// TwinCAT 3 PLC project kfe_rix_motion
// Title: plc-kfe-rix-motion
// Company: SLAC
// ProjectVersion: 2.8.2
// ProgramVersion: 3.1.4022.7
// CompilerDefines: K
// libraries:
//   LCLS General, * (SLAC)
//   lcls-twincat-common-components, * (SLAC)
//   lcls-twincat-motion, * (SLAC)
//   lcls-twincat-physics, * (SLAC)
//   PMPS, * (SLAC - LCLS)
//   Tc2_Standard, * (Beckhoff Automation GmbH)
//   Tc2_System, * (Beckhoff Automation GmbH)
//   Tc3_Module, * (Beckhoff Automation GmbH)
// project tree:
//   DUTs/ DUT_SATT_Filter.TcDUT, ENUM_SXR_SATT_Position.TcDUT
//   Version/ Global_Version.TcGVL
//   GVLs/ GVL.TcGVL, Main.TcGVL
//   / PlcTask.TcTTO
//   POUs/ PRG_1_PlcTask.TcPOU, PRG_2_PMPS_PRE.TcPOU, PRG_3_PMPS_POST.TcPOU, PRG_4_LOG.TcPOU, PRG_AT1K2_SOLID.TcPOU, PRG_AT2K2_SOLID.TcPOU, PRG_AT3K2_SOLID.TcPOU, PRG_IM6K2_PPM.TcPOU, PRG_LI3K2_K2B.TcPOU, PRG_PF1K2_WFS.TcPOU, PRG_LI2K2_K2A.TcPOU, PRG_IM1K1_PPM.TcPOU, PRG_AL1K2_L2SI.TcPOU, PRG_IM2K2_PPM.TcPOU, PRG_IM2K1_PPM.TcPOU, PRG_IM1K2_PPM.TcPOU, PRG_IM3K2_PPM.TcPOU, PRG_IM4K2_PPM.TcPOU, PRG_IM5K2_PPM.TcPOU, PRG_PF2K2_WFS.TcPOU, PRG_SP1K2_PAX.TcPOU, PRG_SP2K2_TXAS.TcPOU, PRG_TM1K2_ATM.TcPOU, PRG_TM2K2_ATM.TcPOU, PRG_ST3K2_TERM.TcPOU
//   POUs/TM1K2/ E_TM1K2_States.TcDUT, FB_TM1K2.TcPOU
//   POUs/TM2K2/ E_TM2K2_States.TcDUT, FB_TM2K2.TcPOU
// real-time tasks:
//   TASK PlcTask: cycle T#10ms, priority 20, ADS port 350
// motion (NC):
//   TASK NC-Task 1 SAF: cycle T#1ms, priority 4, ADS port 501
//   TASK NC-Task 1 SVB: cycle T#10ms, priority 8, ADS port 511
//   AXIS Axis 1 IM1K1-PPM-MMS (id 1)
//     Dynamic: AccelerationMaximum=200, DecelerationMaximum=200, Acceleration=200, Deceleration=200, Jerk=1000, DelayTime=0.004
//     Velo: Maximum=65
//     MotionControl: Enable=true, Range=0.0005, Time=1
//     TargetPosControl: Range=0.01, Time=1
//     OtherSettings: AllowMotionCmdToSlave=true
//     encoder EncType=29
//       EncPara: ScaleFactorNumerator=5e-05, Offset=-214686.941, MaxCount=#xffffffff, ReferenceSystem=1
//         SoftEndMinControl: Enable=true, Range=-100
//         SoftEndMaxControl: Enable=true, Range=-8.82
//         Inc: RefSoftSyncMask=#x0000ffff
//     drive DrvType=24
//       Analog: VeloReferenz=100, ScaleFactorActTorque=0.1
//       TimeComp: TaskDelayCycles=1
//     controller CtrType=2
//       CtrPara: PriorControlFactor=1
//         PosDiffControl: Range=10, Time=0.1
//         PID: PosKp=10, PosExtKp=0.01, PosExtVelo=0.0005, DeadBandPosition=0.0001
//         Observer: BandWidth=20
//   AXIS Axis 2 IM2K1-PPM-MMS (id 2)
//     Dynamic: AccelerationMaximum=200, DecelerationMaximum=200, Acceleration=200, Deceleration=200, Jerk=1000, DelayTime=0.004
//     Velo: Maximum=65
//     MotionControl: Enable=true, Range=0.0005, Time=1
//     TargetPosControl: Range=0.01, Time=1
//     OtherSettings: AllowMotionCmdToSlave=true
//     encoder EncType=29
//       EncPara: ScaleFactorNumerator=5e-05, Offset=-214686.941, MaxCount=#xffffffff, ReferenceSystem=1
//         SoftEndMinControl: Enable=true, Range=-100
//         SoftEndMaxControl: Enable=true, Range=-9.09
//         Inc: RefSoftSyncMask=#x0000ffff
//     drive DrvType=24
//       Analog: VeloReferenz=100, ScaleFactorActTorque=0.1
//       TimeComp: TaskDelayCycles=1
//     controller CtrType=2
//       CtrPara: PriorControlFactor=1
//         PosDiffControl: Range=10, Time=0.1
//         PID: PosKp=10, PosExtKp=0.01, PosExtVelo=0.0005, DeadBandPosition=0.0001
//         Observer: BandWidth=20
//   AXIS Axis 3 SPARE (id 3)
//     Velo: RefSearch=0.1, RefSync=0.1, SlowManual=0.1, FastManual=1, Maximum=1
//     OtherSettings: AllowMotionCmdToSlave=true, PulseDistancePos=1, PulseDistanceNeg=1
//     encoder EncType=29
//       EncPara: ScaleFactorNumerator=1e-06, Offset=-4264.0407, MaxCount=#xffffffff, ReferenceSystem=1
//         SoftEndMinControl: Enable=true
//         SoftEndMaxControl: Enable=true, Range=12.192
//         Inc: RefSoftSyncMask=#x0000ffff
//     drive DrvType=24
//       Analog: VeloReferenz=3.175, ScaleFactorActTorque=0.1
//       TimeComp: TaskDelayCycles=1
//     controller CtrType=1
//       CtrPara: PriorControlFactor=1
//         PosDiffControl: Range=0.1
//         Observer: BandWidth=20
//   AXIS Axis 4 IM1K2-PPM-MMS (id 4)
//     Dynamic: AccelerationMaximum=200, DecelerationMaximum=200, Acceleration=200, Deceleration=200, Jerk=500, DelayTime=0.004
//     Velo: Maximum=65
//     TargetPosControl: Range=0.002, Time=2
//     OtherSettings: AllowMotionCmdToSlave=true
//     encoder EncType=29
//       EncPara: ScaleFactorNumerator=5e-05, Offset=-214686.941, MaxCount=#xffffffff, ReferenceSystem=1
//         SoftEndMinControl: Enable=true, Range=-101
//         SoftEndMaxControl: Enable=true, Range=-9
//         Inc: RefSoftSyncMask=#x0000ffff
//     drive DrvType=24
//       Analog: VeloReferenz=100, ScaleFactorActTorque=0.1
//       TimeComp: TaskDelayCycles=1
//     controller CtrType=2
//       CtrPara: PriorControlFactor=1
//         PosDiffControl: Range=1
//         PID: PosKp=20, PosExtKp=1, PosExtVelo=0.1, DeadBandPosition=0.002
//         Observer: BandWidth=20
//   AXIS Axis 9 TM1K2-MMS-Y (id 9)
//     Dynamic: AccelerationMaximum=200, DecelerationMaximum=200, Acceleration=10, Deceleration=10, Jerk=500, DelayTime=0.004
//     Velo: Maximum=20
//     TargetPosControl: Range=0.002, Time=2
//     OtherSettings: AllowMotionCmdToSlave=true
//     encoder EncType=29
//       EncPara: ScaleFactorNumerator=5e-05, Offset=-214702, MaxCount=#xffffffff, ReferenceSystem=1
//         SoftEndMinControl: Range=-100
//         SoftEndMaxControl: Range=-16
//         Inc: RefSoftSyncMask=#x0000ffff
//     drive DrvType=24
//       Analog: VeloReferenz=100, ScaleFactorActTorque=0.1
//       TimeComp: TaskDelayCycles=1
//     controller CtrType=2
//       CtrPara: PriorControlFactor=1
//         PosDiffControl: Range=1
//         PID: PosKp=20, PosExtKp=1, PosExtVelo=0.1, DeadBandPosition=0.002
//         Observer: BandWidth=20
//   AXIS Axis 10 TM1K2-MMS-X (id 10)
//     Dynamic: AccelerationMaximum=200, DecelerationMaximum=200, Acceleration=10, Deceleration=50, Jerk=500
//     Velo: Maximum=5
//     OtherSettings: AllowMotionCmdToSlave=true
//     encoder EncType=29
//       EncPara: ScaleFactorNumerator=5e-05, MaxCount=#xffffffff, ReferenceSystem=1
//         SoftEndMinControl: Range=8.1
//         SoftEndMaxControl: Range=12.5
//         Inc: RefSoftSyncMask=#x0000ffff
//     drive DrvType=24
//       Analog: VeloReferenz=15.875, ScaleFactorActTorque=0.1
//       TimeComp: TaskDelayCycles=1
//     controller CtrType=1
//       CtrPara: PriorControlFactor=1
//         PosDiffControl: Range=0.2
//         Observer: BandWidth=20
//   AXIS Axis 6 IM2K2-PPM-MMS (id 6)
//     Dynamic: AccelerationMaximum=200, DecelerationMaximum=200, Acceleration=200, Deceleration=200, Jerk=500, DelayTime=0.004
//     Velo: Maximum=65
//     TargetPosControl: Range=0.002, Time=2
//     OtherSettings: AllowMotionCmdToSlave=true
//     encoder EncType=29
//       EncPara: ScaleFactorNumerator=5e-05, Offset=-214686.941, MaxCount=#xffffffff, ReferenceSystem=1
//         SoftEndMinControl: Enable=true, Range=-99
//         SoftEndMaxControl: Enable=true, Range=-7
//         Inc: RefSoftSyncMask=#x0000ffff
//     drive DrvType=24
//       Analog: VeloReferenz=100, ScaleFactorActTorque=0.1
//       TimeComp: TaskDelayCycles=1
//     controller CtrType=2
//       CtrPara: PriorControlFactor=1
//         PosDiffControl: Range=1
//         PID: PosKp=20, PosExtKp=1, PosExtVelo=0.1, DeadBandPosition=0.002
//         Observer: BandWidth=20
//   AXIS Axis 7 IM3K2-PPM-MMS (id 7)
//     Dynamic: AccelerationMaximum=200, DecelerationMaximum=200, Acceleration=200, Deceleration=200, Jerk=500, DelayTime=0.004
//     Velo: Maximum=65
//     TargetPosControl: Range=0.002, Time=2
//     OtherSettings: AllowMotionCmdToSlave=true
//     encoder EncType=29
//       EncPara: ScaleFactorNumerator=5e-05, Offset=-214686.941, MaxCount=#xffffffff, ReferenceSystem=1
//         SoftEndMinControl: Enable=true, Range=-108
//         SoftEndMaxControl: Enable=true, Range=-8
//         Inc: RefSoftSyncMask=#x0000ffff
//     drive DrvType=24
//       Analog: VeloReferenz=100, ScaleFactorActTorque=0.1
//       TimeComp: TaskDelayCycles=1
//     controller CtrType=2
//       CtrPara: PriorControlFactor=1
//         PosDiffControl: Range=1
//         PID: PosKp=20, PosExtKp=1, PosExtVelo=0.1, DeadBandPosition=0.002
//         Observer: BandWidth=20
//   AXIS Axis 8 IM4K2-PPM-MMS (id 8)
//     Dynamic: AccelerationMaximum=200, DecelerationMaximum=200, Acceleration=200, Deceleration=200, Jerk=1000, DelayTime=0.004
//     Velo: Maximum=65
//     MotionControl: Enable=true, Range=0.0005, Time=1
//     TargetPosControl: Range=0.01, Time=1
//     OtherSettings: AllowMotionCmdToSlave=true
//     encoder EncType=29
//       EncPara: ScaleFactorNumerator=5e-05, Offset=-214686.941, MaxCount=#xffffffff, ReferenceSystem=1
//         SoftEndMinControl: Enable=true, Range=-100
//         SoftEndMaxControl: Enable=true, Range=-10
//         Inc: RefSoftSyncMask=#x0000ffff
//     drive DrvType=24
//       Analog: VeloReferenz=100, ScaleFactorActTorque=0.1
//       TimeComp: TaskDelayCycles=1
//     controller CtrType=2
//       CtrPara: PriorControlFactor=1
//         PosDiffControl: Range=10, Time=0.1
//         PID: PosKp=10, PosExtKp=0.01, PosExtVelo=0.0005, DeadBandPosition=0.0001
//         Observer: BandWidth=20
//   AXIS Axis 14 IM5K2-PPM-MMS (id 14)
//     Dynamic: AccelerationMaximum=200, DecelerationMaximum=200, Acceleration=200, Deceleration=200, Jerk=1000, DelayTime=0.004
//     Velo: Maximum=65
//     MotionControl: Enable=true, Range=0.0005, Time=1
//     TargetPosControl: Range=0.01, Time=1
//     OtherSettings: AllowMotionCmdToSlave=true
//     encoder EncType=29
//       EncPara: ScaleFactorNumerator=5e-05, Offset=-214686.941, MaxCount=#xffffffff, ReferenceSystem=1
//         SoftEndMinControl: Enable=true, Range=-100
//         SoftEndMaxControl: Enable=true, Range=-8
//         Inc: RefSoftSyncMask=#x0000ffff
//     drive DrvType=24
//       Analog: VeloReferenz=100, ScaleFactorActTorque=0.1
//       TimeComp: TaskDelayCycles=1
//     controller CtrType=2
//       CtrPara: PriorControlFactor=1
//         PosDiffControl: Range=10, Time=0.1
//         PID: PosKp=10, PosExtKp=0.01, PosExtVelo=0.0005, DeadBandPosition=0.0001
//         Observer: BandWidth=20
//   AXIS Axis 5 AL1K2-L2SI-MMS (id 5)
//     Dynamic: AccelerationMaximum=200, DecelerationMaximum=200, Acceleration=200, Deceleration=200, Jerk=500, DelayTime=0.004
//     Velo: Maximum=10
//     TargetPosControl: Range=0.002, Time=2
//     OtherSettings: AllowMotionCmdToSlave=true
//     encoder EncType=29
//       EncPara: ScaleFactorNumerator=5e-05, Offset=-214686.941, MaxCount=#xffffffff, ReferenceSystem=1
//         SoftEndMinControl: Range=-108.74
//         SoftEndMaxControl: Range=-33.49
//         Inc: RefSoftSyncMask=#x0000ffff
//     drive DrvType=24
//       Analog: VeloReferenz=100, ScaleFactorActTorque=0.1
//       TimeComp: TaskDelayCycles=1
//     controller CtrType=2
//       CtrPara: PriorControlFactor=1
//         PosDiffControl: Range=1
//         PID: PosKp=20, PosExtKp=1, PosExtVelo=0.1, DeadBandPosition=0.002
//         Observer: BandWidth=20
//   AXIS Axis 11 LI2K2-K2A_OUT-MMS (id 11)
//     Dynamic: AccelerationMaximum=200, DecelerationMaximum=200, Acceleration=200, Deceleration=200, Jerk=500, DelayTime=0.004
//     Velo: Maximum=65
//     TargetPosControl: Range=0.002, Time=2
//     OtherSettings: AllowMotionCmdToSlave=true
//     encoder EncType=29
//       EncPara: ScaleFactorNumerator=5e-05, Offset=-214680, MaxCount=#xffffffff, ReferenceSystem=1
//         SoftEndMinControl: Range=-107.43
//         SoftEndMaxControl: Range=1.35
//         Inc: RefSoftSyncMask=#x0000ffff
//     drive DrvType=24
//       Analog: VeloReferenz=100, ScaleFactorActTorque=0.1
//       TimeComp: TaskDelayCycles=1
//     controller CtrType=2
//       CtrPara: PriorControlFactor=1
//         PosDiffControl: Range=1
//         PID: PosKp=20, PosExtKp=1, PosExtVelo=0.1, DeadBandPosition=0.002
//         Observer: BandWidth=20
//   AXIS Axis 12 PF1K2-WFS-MMS-Y (id 12)
//     Dynamic: AccelerationMaximum=200, DecelerationMaximum=200, Acceleration=10, Deceleration=10, Jerk=500, DelayTime=0.004
//     Velo: Maximum=20
//     TargetPosControl: Range=0.002, Time=2
//     OtherSettings: AllowMotionCmdToSlave=true
//     encoder EncType=29
//       EncPara: ScaleFactorNumerator=5e-05, Offset=-214679, MaxCount=#xffffffff, ReferenceSystem=1
//         SoftEndMinControl: Enable=true, Range=-94
//         SoftEndMaxControl: Enable=true, Range=-9.71
//         Inc: RefSoftSyncMask=#x0000ffff
//     drive DrvType=24
//       Analog: VeloReferenz=100, ScaleFactorActTorque=0.1
//       TimeComp: TaskDelayCycles=1
//     controller CtrType=2
//       CtrPara: PriorControlFactor=1
//         PosDiffControl: Range=1
//         PID: PosKp=20, PosExtKp=1, PosExtVelo=0.1, DeadBandPosition=0.002
//         Observer: BandWidth=20
//   AXIS Axis 13 PF1K2-WFS-MMS-Z (id 13)
//     Dynamic: AccelerationMaximum=200, DecelerationMaximum=200, Acceleration=10, Deceleration=50, Jerk=500
//     Velo: Maximum=5
//     OtherSettings: AllowMotionCmdToSlave=true
//     encoder EncType=29
//       EncPara: ScaleFactorNumerator=5e-05, MaxCount=#xffffffff, ReferenceSystem=1
//         SoftEndMinControl: Range=6.5
//         SoftEndMaxControl: Range=56
//         Inc: RefSoftSyncMask=#x0000ffff
//     drive DrvType=24
//       DrvPara: Inverse=true
//         Analog: VeloReferenz=15.875, ScaleFactorActTorque=0.1
//         TimeComp: TaskDelayCycles=1
//     controller CtrType=1
//       CtrPara: PriorControlFactor=1
//         PosDiffControl: Range=1
//         Observer: BandWidth=20
//   AXIS Axis 15 TM2K2-MMS-Y (id 15)
//     Dynamic: AccelerationMaximum=200, DecelerationMaximum=200, Acceleration=10, Deceleration=10, Jerk=500, DelayTime=0.004
//     Velo: Maximum=20
//     TargetPosControl: Range=0.002, Time=2
//     OtherSettings: AllowMotionCmdToSlave=true
//     encoder EncType=29
//       EncPara: ScaleFactorNumerator=5e-05, Offset=-214682, MaxCount=#xffffffff, ReferenceSystem=1
//         SoftEndMinControl: Range=-100
//         SoftEndMaxControl: Range=-16
//         Inc: RefSoftSyncMask=#x0000ffff
//     drive DrvType=24
//       Analog: VeloReferenz=100, ScaleFactorActTorque=0.1
//       TimeComp: TaskDelayCycles=1
//     controller CtrType=2
//       CtrPara: PriorControlFactor=1
//         PosDiffControl: Range=1
//         PID: PosKp=20, PosExtKp=1, PosExtVelo=0.1, DeadBandPosition=0.002
//         Observer: BandWidth=20
//   AXIS Axis 16 TM2K2-MMS-X (id 16)
//     Dynamic: AccelerationMaximum=200, DecelerationMaximum=200, Acceleration=10, Deceleration=50, Jerk=500
//     Velo: Maximum=5
//     OtherSettings: AllowMotionCmdToSlave=true
//     encoder EncType=29
//       EncPara: ScaleFactorNumerator=5e-05, MaxCount=#xffffffff, ReferenceSystem=1
//         SoftEndMinControl: Enable=true, Range=16.5
//         SoftEndMaxControl: Enable=true, Range=21
//         Inc: RefSoftSyncMask=#x0000ffff
//     drive DrvType=24
//       DrvPara: Inverse=true
//         Analog: VeloReferenz=15.875, ScaleFactorActTorque=0.1
//         TimeComp: TaskDelayCycles=1
//     controller CtrType=1
//       CtrPara: PriorControlFactor=1
//         PosDiffControl: Range=0.2
//         Observer: BandWidth=20
//   AXIS Axis 17 AT2K2-SOLID-MMS-01 (id 17)
//     Dynamic: AccelerationMaximum=400, DecelerationMaximum=400, Acceleration=160, Deceleration=160, Jerk=80, DelayTime=0.008
//     Velo: SlowManual=1, FastManual=10, Maximum=80
//     OtherSettings: AllowMotionCmdToSlave=true
//     encoder EncType=29
//       EncPara: ScaleFactorNumerator=5e-05, MaxCount=#xffffffff
//         SoftEndMinControl: Enable=true, Range=16.5
//         SoftEndMaxControl: Enable=true, Range=152.5
//         Inc: RefSoftSyncMask=#x0000ffff
//     drive DrvType=24
//       Analog: VeloReferenz=40, ScaleFactorActTorque=0.1
//       TimeComp: TaskDelayCycles=1
//     controller CtrType=2
//       CtrPara: PriorControlFactor=1
//         PosDiffControl: Range=0.2
//         PID: PosKp=20, PosExtKp=20, PosExtVelo=0.1, DeadBandPosition=0.01
//         Observer: BandWidth=20
//   AXIS Axis 18 AT2K2-SOLID-MMS-02 (id 18)
//     Dynamic: AccelerationMaximum=400, DecelerationMaximum=400, Acceleration=160, Deceleration=160, Jerk=80, DelayTime=0.008
//     Velo: SlowManual=1, FastManual=5, Maximum=80
//     OtherSettings: AllowMotionCmdToSlave=true
//     encoder EncType=29
//       EncPara: ScaleFactorNumerator=5e-05, MaxCount=#xffffffff
//         SoftEndMinControl: Enable=true, Range=17.5
//         SoftEndMaxControl: Enable=true, Range=152.5
//         Inc: RefSoftSyncMask=#x0000ffff
//     drive DrvType=24
//       Analog: VeloReferenz=40, ScaleFactorActTorque=0.1
//       TimeComp: TaskDelayCycles=1
//     controller CtrType=2
//       CtrPara: PriorControlFactor=1
//         PosDiffControl: Range=0.2
//         PID: PosKp=20, PosExtKp=20, PosExtVelo=0.1, DeadBandPosition=0.01
//         Observer: BandWidth=20
//   AXIS Axis 19 AT2K2-SOLID-MMS-03 (id 19)
//     Dynamic: AccelerationMaximum=400, DecelerationMaximum=400, Acceleration=160, Deceleration=160, Jerk=80, DelayTime=0.008
//     Velo: SlowManual=1, FastManual=10, Maximum=80
//     OtherSettings: AllowMotionCmdToSlave=true
//     encoder EncType=29
//       EncPara: ScaleFactorNumerator=5e-05, MaxCount=#xffffffff
//         SoftEndMinControl: Enable=true, Range=16.5
//         SoftEndMaxControl: Enable=true, Range=152.5
//         Inc: RefSoftSyncMask=#x0000ffff
//     drive DrvType=24
//       Analog: VeloReferenz=40, ScaleFactorActTorque=0.1
//       TimeComp: TaskDelayCycles=1
//     controller CtrType=2
//       CtrPara: PriorControlFactor=1
//         PosDiffControl: Range=0.2
//         PID: PosKp=20, PosExtKp=20, PosExtVelo=0.1, DeadBandPosition=0.01
//         Observer: BandWidth=20
//   AXIS Axis 20 AT2K2-SOLID-MMS-04 (id 20)
//     Dynamic: AccelerationMaximum=400, DecelerationMaximum=400, Acceleration=160, Deceleration=160, Jerk=80, DelayTime=0.008
//     Velo: SlowManual=1, FastManual=10, Maximum=80
//     OtherSettings: AllowMotionCmdToSlave=true
//     encoder EncType=29
//       EncPara: ScaleFactorNumerator=5e-05, MaxCount=#xffffffff
//         SoftEndMinControl: Enable=true, Range=17.8
//         SoftEndMaxControl: Enable=true, Range=152.5
//         Inc: RefSoftSyncMask=#x0000ffff
//     drive DrvType=24
//       Analog: VeloReferenz=40, ScaleFactorActTorque=0.1
//       TimeComp: TaskDelayCycles=1
//     controller CtrType=2
//       CtrPara: PriorControlFactor=1
//         PosDiffControl: Range=0.2
//         PID: PosKp=20, PosExtKp=20, PosExtVelo=0.1, DeadBandPosition=0.01
//         Observer: BandWidth=20
//   AXIS Axis 21 LI3K2-K2B-MMS (id 21)
//     Dynamic: AccelerationMaximum=200, DecelerationMaximum=200, Acceleration=200, Deceleration=200, Jerk=500, DelayTime=0.004
//     Velo: Maximum=65
//     TargetPosControl: Range=0.002, Time=2
//     OtherSettings: AllowMotionCmdToSlave=true
//     encoder EncType=29
//       EncPara: ScaleFactorNumerator=5e-05, Offset=-214687, MaxCount=#xffffffff, ReferenceSystem=1
//         SoftEndMinControl: Enable=true, Range=-107.43
//         SoftEndMaxControl: Enable=true, Range=1.35
//         Inc: RefSoftSyncMask=#x0000ffff
//     drive DrvType=24
//       Analog: VeloReferenz=100, ScaleFactorActTorque=0.1
//       TimeComp: TaskDelayCycles=1
//     controller CtrType=2
//       CtrPara: PriorControlFactor=1
//         PosDiffControl: Range=1
//         PID: PosKp=20, PosExtKp=1, PosExtVelo=0.1, DeadBandPosition=0.002
//         Observer: BandWidth=20
//   AXIS Axis 22 PF2K2-WFS-MMS-Y (id 22)
//     Dynamic: AccelerationMaximum=200, DecelerationMaximum=200, Acceleration=10, Deceleration=10, Jerk=500, DelayTime=0.004
//     Velo: Maximum=20
//     TargetPosControl: Range=0.002, Time=2
//     OtherSettings: AllowMotionCmdToSlave=true
//     encoder EncType=29
//       EncPara: ScaleFactorNumerator=5e-05, Offset=-214687, MaxCount=#xffffffff, ReferenceSystem=1
//         SoftEndMinControl: Enable=true, Range=-99.33
//         SoftEndMaxControl: Enable=true, Range=-9.71
//         Inc: RefSoftSyncMask=#x0000ffff
//     drive DrvType=24
//       Analog: VeloReferenz=100, ScaleFactorActTorque=0.1
//       TimeComp: TaskDelayCycles=1
//     controller CtrType=2
//       CtrPara: PriorControlFactor=1
//         PosDiffControl: Range=1
//         PID: PosKp=20, PosExtKp=1, PosExtVelo=0.1, DeadBandPosition=0.002
//         Observer: BandWidth=20
//   AXIS Axis 23 PF2K2-WFS-MMS-Z (id 23)
//     Dynamic: AccelerationMaximum=200, DecelerationMaximum=200, Acceleration=10, Deceleration=50, Jerk=500
//     Velo: Maximum=5
//     OtherSettings: AllowMotionCmdToSlave=true
//     encoder EncType=29
//       EncPara: ScaleFactorNumerator=5e-05, MaxCount=#xffffffff, ReferenceSystem=1
//         SoftEndMinControl: Range=6.5
//         SoftEndMaxControl: Range=56
//         Inc: RefSoftSyncMask=#x0000ffff
//     drive DrvType=24
//       DrvPara: Inverse=true
//         Analog: VeloReferenz=15.875, ScaleFactorActTorque=0.1
//         TimeComp: TaskDelayCycles=1
//     controller CtrType=1
//       CtrPara: PriorControlFactor=1
//         PosDiffControl: Range=1
//         PID: PosKp=10
//         Observer: BandWidth=20
//   AXIS Axis 24 IM6K2-PPM-MMS (id 24)
//     Dynamic: AccelerationMaximum=200, DecelerationMaximum=200, Acceleration=200, Deceleration=200, Jerk=1000, DelayTime=0.004
//     Velo: Maximum=65
//     MotionControl: Enable=true, Range=0.0005, Time=1
//     TargetPosControl: Range=0.01, Time=1
//     OtherSettings: AllowMotionCmdToSlave=true
//     encoder EncType=29
//       EncPara: ScaleFactorNumerator=5e-05, Offset=-214686.941, MaxCount=#xffffffff, ReferenceSystem=1
//         SoftEndMinControl: Enable=true, Range=-100
//         SoftEndMaxControl: Enable=true, Range=-8
//         Inc: RefSoftSyncMask=#x0000ffff
//     drive DrvType=24
//       Analog: VeloReferenz=100, ScaleFactorActTorque=0.1
//       TimeComp: TaskDelayCycles=1
//     controller CtrType=2
//       CtrPara: PriorControlFactor=1
//         PosDiffControl: Range=10, Time=0.1
//         PID: PosKp=10, PosExtKp=0.01, PosExtVelo=0.0005, DeadBandPosition=0.0001
//         Observer: BandWidth=20
//   AXIS Axis 25 AT1K2-SOLID-MMS-01 (id 25)
//     Dynamic: AccelerationMaximum=400, DecelerationMaximum=400, Acceleration=160, Deceleration=160, Jerk=80, DelayTime=0.008
//     Velo: SlowManual=1, FastManual=10, Maximum=80
//     OtherSettings: AllowMotionCmdToSlave=true
//     encoder EncType=29
//       EncPara: ScaleFactorNumerator=5e-05, MaxCount=#xffffffff
//         SoftEndMinControl: Enable=true, Range=19
//         SoftEndMaxControl: Enable=true, Range=152.2
//         Inc: RefSoftSyncMask=#x0000ffff
//     drive DrvType=24
//       Analog: VeloReferenz=40, ScaleFactorActTorque=0.1
//       TimeComp: TaskDelayCycles=1
//     controller CtrType=2
//       CtrPara: PriorControlFactor=1
//         PosDiffControl: Range=0.2
//         PID: PosKp=20, PosExtKp=20, PosExtVelo=0.1, DeadBandPosition=0.01
//         Observer: BandWidth=20
//   AXIS Axis 26 AT1K2-SOLID-MMS-02 (id 26)
//     Dynamic: AccelerationMaximum=400, DecelerationMaximum=400, Acceleration=160, Deceleration=160, Jerk=80, DelayTime=0.008
//     Velo: SlowManual=1, FastManual=10, Maximum=80
//     OtherSettings: AllowMotionCmdToSlave=true
//     encoder EncType=29
//       EncPara: ScaleFactorNumerator=5e-05, MaxCount=#xffffffff
//         SoftEndMinControl: Enable=true, Range=19
//         SoftEndMaxControl: Enable=true, Range=152.2
//         Inc: RefSoftSyncMask=#x0000ffff
//     drive DrvType=24
//       Analog: VeloReferenz=40, ScaleFactorActTorque=0.1
//       TimeComp: TaskDelayCycles=1
//     controller CtrType=2
//       CtrPara: PriorControlFactor=1
//         PosDiffControl: Range=0.2
//         PID: PosKp=20, PosExtKp=20, PosExtVelo=0.1, DeadBandPosition=0.01
//         Observer: BandWidth=20
//   AXIS Axis 27 AT1K2-SOLID-MMS-03 (id 27)
//     Dynamic: AccelerationMaximum=400, DecelerationMaximum=400, Acceleration=160, Deceleration=160, Jerk=80, DelayTime=0.008
//     Velo: SlowManual=1, FastManual=10, Maximum=6
//     OtherSettings: AllowMotionCmdToSlave=true
//     encoder EncType=29
//       EncPara: ScaleFactorNumerator=5e-05, MaxCount=#xffffffff
//         SoftEndMinControl: Enable=true, Range=23
//         SoftEndMaxControl: Enable=true, Range=67
//         Inc: RefSoftSyncMask=#x0000ffff
//     drive DrvType=24
//       Analog: VeloReferenz=2.5, ScaleFactorActTorque=0.1
//       TimeComp: TaskDelayCycles=1
//     controller CtrType=2
//       CtrPara: PriorControlFactor=1
//         PosDiffControl: Range=0.2
//         PID: PosKp=5, PosExtKp=5, PosExtVelo=0.1, DeadBandPosition=0.001
//         Observer: BandWidth=20
//   AXIS Axis 37 SP1K2-PAX-BB-MMS-Y-02 (id 37)
//     Velo: SlowManual=0.5, FastManual=1, Maximum=1.5
//     OtherSettings: AllowMotionCmdToSlave=true
//     encoder EncType=29
//       EncPara: ScaleFactorNumerator=0.000244, Offset=-8917.43869, MaxCount=#xffffffff
//         SoftEndMinControl: Enable=true
//         SoftEndMaxControl: Enable=true, Range=43
//         Inc: RefSoftSyncMask=#x0000ffff
//     drive DrvType=24
//       DrvPara: Inverse=true
//         Analog: VeloReferenz=2.5, ScaleFactorActTorque=0.1
//         TimeComp: TaskDelayCycles=1
//     controller CtrType=1
//       CtrPara: PriorControlFactor=1
//         Observer: BandWidth=20
//   AXIS Axis 36 SP1K2-PAX-BB-MMS-Y-01 (id 36)
//     Velo: SlowManual=0.5, FastManual=1, Maximum=1.5
//     OtherSettings: AllowMotionCmdToSlave=true
//     encoder EncType=29
//       EncPara: ScaleFactorNumerator=0.000244, Offset=-1039158.545, MaxCount=#xffffffff
//         SoftEndMinControl: Enable=true, Range=-43
//         SoftEndMaxControl: Enable=true
//         Inc: RefSoftSyncMask=#x0000ffff
//     drive DrvType=24
//       Analog: VeloReferenz=2.5, ScaleFactorActTorque=0.1
//       TimeComp: TaskDelayCycles=1
//     controller CtrType=1
//       CtrPara: PriorControlFactor=1
//         Observer: BandWidth=20
//   AXIS Axis 35 SP1K2-PAX-TAR-MMS-RY (id 35)
//     OtherSettings: AllowMotionCmdToSlave=true
//     encoder EncType=1
//       Inc: RefSoftSyncMask=#x0000ffff
//     drive DrvType=5
//       Analog: ScaleFactorActTorque=0.1
//       TimeComp: TaskDelayCycles=1
//     controller CtrType=1
//       CtrPara: PriorControlFactor=1
//         Observer: BandWidth=20
//   AXIS Axis 34 SP1K2-PAX-TAR-MMS-Z (id 34)
//     Velo: SlowManual=0.1, FastManual=1, Maximum=1
//     OtherSettings: AllowMotionCmdToSlave=true
//     encoder EncType=29
//       EncPara: ScaleFactorNumerator=0.000244, Offset=-15736.2402, MaxCount=#xffffffff
//         SoftEndMinControl: Enable=true
//         Inc: RefSoftSyncMask=#x0000ffff
//     drive DrvType=24
//       Analog: VeloReferenz=2, ScaleFactorActTorque=0.1
//       TimeComp: TaskDelayCycles=1
//     controller CtrType=1
//       CtrPara: PriorControlFactor=1
//         Observer: BandWidth=20
//   AXIS Axis 33 SP1K2-PAX-TAR-MMS-Y (id 33)
//     Velo: SlowManual=0.5, FastManual=1, Maximum=1
//     OtherSettings: AllowMotionCmdToSlave=true
//     encoder EncType=29
//       EncPara: ScaleFactorNumerator=5e-05, MaxCount=#xffffffff
//         Inc: RefSoftSyncMask=#x0000ffff
//     drive DrvType=24
//       DrvPara: Inverse=true
//         Analog: VeloReferenz=2, ScaleFactorActTorque=0.1
//         TimeComp: TaskDelayCycles=1
//     controller CtrType=1
//       CtrPara: PriorControlFactor=1
//         Observer: BandWidth=20
//   AXIS Axis 32 SP1K2-PAX-TAR-MMS-X (id 32)
//     Dynamic: AccelerationMaximum=1, DecelerationMaximum=1
//     Velo: SlowManual=0.1, FastManual=1, Maximum=0.5
//     OtherSettings: AllowMotionCmdToSlave=true
//     encoder EncType=29
//       EncPara: ScaleFactorNumerator=0.000244, Offset=-15554.7601, MaxCount=#xffffffff
//         Inc: RefSoftSyncMask=#x0000ffff
//     drive DrvType=24
//       DrvPara: Inverse=true
//         Analog: VeloReferenz=12.5, ScaleFactorActTorque=0.1
//         TimeComp: TaskDelayCycles=1
//     controller CtrType=1
//       CtrPara: PriorControlFactor=1
//         Observer: BandWidth=20
//   AXIS Axis 31 SP1K2-PAX-FRAME-MMS-X (id 31)
//     Dynamic: AccelerationMaximum=1500
//     Velo: Maximum=1
//     OtherSettings: AllowMotionCmdToSlave=true
//     encoder EncType=29
//       EncPara: ScaleFactorNumerator=5e-05, MaxCount=#xffffffff
//         Inc: RefSoftSyncMask=#x0000ffff
//     drive DrvType=24
//       Analog: VeloReferenz=10, ScaleFactorActTorque=0.1
//       TimeComp: TaskDelayCycles=1
//     controller CtrType=1
//       CtrPara: PriorControlFactor=1
//         Observer: BandWidth=20
//   AXIS Axis 30 SP1K2-PAX-FRAME-MMS-Y-03 (id 30)
//     Velo: Maximum=1
//     OtherSettings: AllowMotionCmdToSlave=true
//     encoder EncType=29
//       EncPara: ScaleFactorNumerator=5e-05, MaxCount=#xffffffff
//         Inc: RefSoftSyncMask=#x0000ffff
//     drive DrvType=24
//       Analog: VeloReferenz=2.5, ScaleFactorActTorque=0.1
//       TimeComp: TaskDelayCycles=1
//     controller CtrType=1
//       CtrPara: PriorControlFactor=1
//         Observer: BandWidth=20
//   AXIS Axis 29 SP1K2-PAX-FRAME-MMS-Y-02 (id 29)
//     Velo: Maximum=1
//     OtherSettings: AllowMotionCmdToSlave=true
//     encoder EncType=29
//       EncPara: ScaleFactorNumerator=5e-05, MaxCount=#xffffffff
//         Inc: RefSoftSyncMask=#x0000ffff
//     drive DrvType=24
//       Analog: VeloReferenz=2.5, ScaleFactorActTorque=0.1
//       TimeComp: TaskDelayCycles=1
//     controller CtrType=1
//       CtrPara: PriorControlFactor=1
//         Observer: BandWidth=20
//   AXIS Axis 28 SP1K2-PAX-FRAME-MMS-Y-01 (id 28)
//     Velo: Maximum=1
//     OtherSettings: AllowMotionCmdToSlave=true
//     encoder EncType=29
//       EncPara: ScaleFactorNumerator=5e-06, MaxCount=#xffffffff
//         Inc: RefSoftSyncMask=#x0000ffff
//     drive DrvType=24
//       Analog: VeloReferenz=2.5, ScaleFactorActTorque=0.1
//       TimeComp: TaskDelayCycles=1
//     controller CtrType=1
//       CtrPara: PriorControlFactor=1
//         Observer: BandWidth=20
// I/O:
//   DEVICE PLC Rail (EtherCAT), AmsNetId 172.21.140.70.2.1
//     Power (EK1200) [EK1200-5000 EtherCAT Power supply (2A E-Bus)]
//       License (EL6070)
//       PMPS_FFO [EL2202 2Ch. Dig. Output 24V, 0.5A]
//       PMPS_PRE [EL6695 EtherCAT Bridge terminal (Primary)]
//       Fiber Coupler (EK1521-0010) [EK1521-0010 1 port EtherCAT junction (FX-SingleMode)]
//         Term 34 (EK1501-0010) [EK1501-0010 EtherCAT Coupler (2A E-Bus, FX-SingleMode, ID switch)]
//           Term 35 (EL9410) [EL9410 E-Bus Power Supplier  (Diagnostics)]
//           Term 36 (EL2202) [EL2202 2Ch. Dig. Output 24V, 0.5A]
//           Term 37 (EL6070) [EL6070 1Ch. Licensing-Terminal]
//           Term 38 (EL6695) [EL6695 EtherCAT Bridge terminal (Primary)]
//           Term 39 (EK1122) [EK1122 2 port EtherCAT junction]
//             IM1K2-PPM (EK1100) [EK1100 EtherCAT Coupler (2A E-Bus)]
//               IM1K2-EL7041-E1 [EL7041 1Ch. Stepper motor output stage (50V, 5A)]
//               IM1K2-EL5042-E2 [EL5042 2Ch. BiSS-C Encoder]
//               IM1K2-EL2004-E3 [EL2004 4Ch. Dig. Output 24V, 0.5A]
//               IM1K2-EL3314-E4 [EL3314 4Ch. Ana. Input Thermocouple (TC)]
//               IM1K2-EL3052-E5 [EL3052 2Ch. Ana. Input 4-20mA]
//               IM1K2-EL3062-E6 [EL3062 2Ch. Ana. Input 0-10V]
//               IM1K2-EL4004-E7 [EL4004 4Ch. Ana. Output 0-10V, 12bit]
//               IM1K2-EL9011-E8 [EL9011 End Terminal]
//             AL1K2-L2SI (EK1100) [EK1100 EtherCAT Coupler (2A E-Bus)]
//               AL1K2-EL7041-E1 [EL7041 1Ch. Stepper motor output stage (50V, 5A)]
//               AL1K2-EL5042-E2 [EL5042 2Ch. BiSS-C Encoder]
//               AL1K2-EL2004-E3 [EL2004 4Ch. Dig. Output 24V, 0.5A]
//               AL1K2-EL4004-E4 [EL4004 4Ch. Ana. Output 0-10V, 12bit]
//               AL1K2-EL9011-E5 [EL9011 End Terminal]
//           Term 49 (EK1122) [EK1122 2 port EtherCAT junction]
//             IM2K2-PPM (EK1100) [EK1100 EtherCAT Coupler (2A E-Bus)]
//               IM2K2-EL7041-E1 [EL7041 1Ch. Stepper motor output stage (50V, 5A)]
//               IM2K2-EL5042-E2 [EL5042 2Ch. BiSS-C Encoder]
//               IM2K2-EL2004-E3 [EL2004 4Ch. Dig. Output 24V, 0.5A]
//               IM2K2-EL3314-E4 [EL3314 4Ch. Ana. Input Thermocouple (TC)]
//               IM2K2-EL3052-E5 [EL3052 2Ch. Ana. Input 4-20mA]
//               IM2K2-EL3062-E6 [EL3062 2Ch. Ana. Input 0-10V]
//               IM2K2-EL4004-E7 [EL4004 4Ch. Ana. Output 0-10V, 12bit]
//               IM2K2-EL9011-E8
//           Term 50 (EK1122) [EK1122 2 port EtherCAT junction]
//             IM3K2-PPM (EK1100) [EK1100 EtherCAT Coupler (2A E-Bus)]
//               IM3K2-EL7041-E1 [EL7041 1Ch. Stepper motor output stage (50V, 5A)]
//               IM3K2-EL5042-E2 [EL5042 2Ch. BiSS-C Encoder]
//               IM3K2-EL2004-E3 [EL2004 4Ch. Dig. Output 24V, 0.5A]
//               IM3K2-EL3314-E4 [EL3314 4Ch. Ana. Input Thermocouple (TC)]
//               IM3K2-EL3052-E5 [EL3052 2Ch. Ana. Input 4-20mA]
//               IM3K2-EL3062-E6 [EL3062 2Ch. Ana. Input 0-10V]
//               IM3K2-EL4004-E7 [EL4004 4Ch. Ana. Output 0-10V, 12bit]
//               IM3K2-EL9011-E8
//             IM4K2-PPM (EK1100) [EK1100 EtherCAT Coupler (2A E-Bus)]
//               IM4K2-EL7041-E1 [EL7041 1Ch. Stepper motor output stage (50V, 5A)]
//               IM4K2-EL5042-E2 [EL5042 2Ch. BiSS-C Encoder]
//               IM4K2-EL2004-E3 [EL2004 4Ch. Dig. Output 24V, 0.5A]
//               IM4K2-EL3314-E4 [EL3314 4Ch. Ana. Input Thermocouple (TC)]
//               IM4K2-EL3052-E5 [EL3052 2Ch. Ana. Input 4-20mA]
//               IM4K2-EL3062-E6 [EL3062 2Ch. Ana. Input 0-10V]
//               IM4K2-EL4004-E7 [EL4004 4Ch. Ana. Output 0-10V, 12bit]
//               IM4K2-EL3602-0002-E8 [EL3602-0002 2Ch. Ana. Input +/-200mV, Diff. 24bit]
//               IM4K2-EL9011-E9 [EL9011 End Terminal]
//           Term 51 (EK1110)
//         Term 123 (EK1100) [EK1100 EtherCAT Coupler (2A E-Bus)]
//           Term 124 (EK1122) [EK1122 2 port EtherCAT junction]
//             TM1K2-K2A (EK1100) [EK1100 EtherCAT Coupler (2A E-Bus)]
//               TM1K2-EL7041-E1 [EL7041 1Ch. Stepper motor output stage (50V, 5A)]
//               TM1K2-EL7041-E2 [EL7041 1Ch. Stepper motor output stage (50V, 5A)]
//               TM1K2-EL5042-E3 [EL5042 2Ch. BiSS-C Encoder]
//               TM1K2-EL2004-E4 [EL2004 4Ch. Dig. Output 24V, 0.5A]
//               TM1K2-EL3314-E5 [EL3314 4Ch. Ana. Input Thermocouple (TC)]
//               TM1K2-EL9011-E6 [EL9011 End Terminal]
//           Term 131 (EK1122) [EK1122 2 port EtherCAT junction]
//             LI2K2-K2A_OUT  (EK1100) [EK1100 EtherCAT Coupler (2A E-Bus)]
//               LI2K2-EL7041-E1 [EL7041 1Ch. Stepper motor output stage (50V, 5A)]
//               LI2K2-EL2004-E2 [EL2004 4Ch. Dig. Output 24V, 0.5A]
//               LI2K2-EL5042-E3 [EL5042 2Ch. BiSS-C Encoder]
//               LI2K2-EL9011-E4 [EL9011 End Terminal]
//             PF1K2-WFS (EK1100) [EK1100 EtherCAT Coupler (2A E-Bus)]
//               PF1K2-EL7041-E1 [EL7041 1Ch. Stepper motor output stage (50V, 5A)]
//               PF1K2-EL7041-E2 [EL7041 1Ch. Stepper motor output stage (50V, 5A)]
//               PF1K2-EL5042-E3 [EL5042 2Ch. BiSS-C Encoder]
//               PF1K2-EL2004-E4 [EL2004 4Ch. Dig. Output 24V, 0.5A]
//               PF1K2-EL3314-E5 [EL3314 4Ch. Ana. Input Thermocouple (TC)]
//               PF1K2-EL9011-E6 [EL9011 End Terminal]
//           Term 140 (EK1122) [EK1122 2 port EtherCAT junction]
//             IM5K2-PPM (EK1100) [EK1100 EtherCAT Coupler (2A E-Bus)]
//               IM5K2-EL7041-E1 [EL7041 1Ch. Stepper motor output stage (50V, 5A)]
//               IM5K2-EL5042-E2 [EL5042 2Ch. BiSS-C Encoder]
//               IM5K2-EL2004-E3 [EL2004 4Ch. Dig. Output 24V, 0.5A]
//               IM5K2-EL3314-E4 [EL3314 4Ch. Ana. Input Thermocouple (TC)]
//               IM5K2-EL3052-E5 [EL3052 2Ch. Ana. Input 4-20mA]
//               IM5K2-EL3062-E6 [EL3062 2Ch. Ana. Input 0-10V]
//               IM5K2-EL4004-E7 [EL4004 4Ch. Ana. Output 0-10V, 12bit]
//               IM5K2-EL9011-E8 [EL9011 End Terminal]
//             TM2K2-K2B (EK1100) [EK1100 EtherCAT Coupler (2A E-Bus)]
//               TM2K2-EL7041-E1 [EL7041 1Ch. Stepper motor output stage (50V, 5A)]
//               TM2K2-EL7041-E2 [EL7041 1Ch. Stepper motor output stage (50V, 5A)]
//               TM2K2-EL5042-E3 [EL5042 2Ch. BiSS-C Encoder]
//               TM2K2-EL2004-E4 [EL2004 4Ch. Dig. Output 24V, 0.5A]
//               TM2K2-EL3314-E5 [EL3314 4Ch. Ana. Input Thermocouple (TC)]
//               TM2K2-EL3052-E6 [EL3052 2Ch. Ana. Input 4-20mA]
//               TM2K2-EL9011-E7 [EL9011 End Terminal]
//           Term 155 (EK1122) [EK1122 2 port EtherCAT junction]
//             AT2K2-SOLID (EK1100) [EK1100 EtherCAT Coupler (2A E-Bus)]
//               AT2K2-EL7047-01 [EL7047 1Ch. Stepper motor output stage (50V, 5A)]
//               AT2K2-EL7047-02 [EL7047 1Ch. Stepper motor output stage (50V, 5A)]
//               AT2K2-EL7047-03 [EL7047 1Ch. Stepper motor output stage (50V, 5A)]
//               AT2K2-EL7047-04 [EL7047 1Ch. Stepper motor output stage (50V, 5A)]
//               AT2K2-EL5042-01 [EL5042 2Ch. BiSS-C Encoder]
//               AT2K2-EL5042-02 [EL5042 2Ch. BiSS-C Encoder]
//               AT2K2-EL3202-01 [EL3202-0020 2Ch. Ana. Input PT100 (RTD), High Precision, calibrated]
//               AT2K2-EL3202-02 [EL3202-0020 2Ch. Ana. Input PT100 (RTD), High Precision, calibrated]
//               AT2K2-EL3202-03 [EL3202-0020 2Ch. Ana. Input PT100 (RTD), High Precision, calibrated]
//               AT2K2-EL3202-04 [EL3202-0020 2Ch. Ana. Input PT100 (RTD), High Precision, calibrated]
//               AT2K2-EL9011 [EL9011 End Terminal]
//             LI3K2-K2B (EK1100) [EK1100 EtherCAT Coupler (2A E-Bus)]
//               LI3K2-EL7041-E1 [EL7041 1Ch. Stepper motor output stage (50V, 5A)]
//               LI3K2-EL5042-E2 [EL5042 2Ch. BiSS-C Encoder]
//               LI3K2-EL2004-E3 [EL2004 4Ch. Dig. Output 24V, 0.5A]
//               LI3K2-EL3314-E4 [EL3314 4Ch. Ana. Input Thermocouple (TC)]
//               LI3K2-EL3052-E5 [EL3052 2Ch. Ana. Input 4-20mA]
//               LI3K2-EL3062-E6 [EL3062 2Ch. Ana. Input 0-10V]
//               LI3K2-EL4004-E7 [EL4004 4Ch. Ana. Output 0-10V, 12bit]
//               LI3K2-EL9011-E8 [EL9011 End Terminal]
//           Term 156 (EK1122) [EK1122 2 port EtherCAT junction]
//             PF2K2-WFS (EK1100) [EK1100 EtherCAT Coupler (2A E-Bus)]
//               PF2K2-EL7041-E1 [EL7041 1Ch. Stepper motor output stage (50V, 5A)]
//               PF2K2-EL7041-E2 [EL7041 1Ch. Stepper motor output stage (50V, 5A)]
//               PF2K2-EL5042-E3 [EL5042 2Ch. BiSS-C Encoder]
//               PF2K2-EL2004-E4 [EL2004 4Ch. Dig. Output 24V, 0.5A]
//               PF2K2-EL3314-E5 [EL3314 4Ch. Ana. Input Thermocouple (TC)]
//               PF2K2-EL9011-E6 [EL9011 End Terminal]
//             IM6K2-PPM (EK1100) [EK1100 EtherCAT Coupler (2A E-Bus)]
//               IM6K2-EL7041-E1 [EL7041 1Ch. Stepper motor output stage (50V, 5A)]
//               IM6K2-EL5042-E2 [EL5042 2Ch. BiSS-C Encoder]
//               IM6K2-EL2004-E3 [EL2004 4Ch. Dig. Output 24V, 0.5A]
//               IM6K2-EL3314-E4 [EL3314 4Ch. Ana. Input Thermocouple (TC)]
//               IM6K2-EL3052-E5 [EL3052 2Ch. Ana. Input 4-20mA]
//               IM6K2-EL3062-E6 [EL3062 2Ch. Ana. Input 0-10V]
//               IM6K2-EL4004-E7 [EL4004 4Ch. Ana. Output 0-10V, 12bit]
//               IM6K2-EL3602-E8 [EL3602 2Ch. Ana. Input +/-10Volt, Diff. 24bit]
//               IM6K2-EL9011-E9 [EL9011 End Terminal]
//           Term 157 (EK1122) [EK1122 2 port EtherCAT junction]
//             AT1K2-SOLID (EK1100) [EK1100 EtherCAT Coupler (2A E-Bus)]
//               AT1K2-EL7047-01 [EL7047 1Ch. Stepper motor output stage (50V, 5A)]
//               AT1K2-EL7047-02 [EL7047 1Ch. Stepper motor output stage (50V, 5A)]
//               AT1K2-EL7047-03 [EL7047 1Ch. Stepper motor output stage (50V, 5A)]
//               AT1K2-EL5042-01 [EL5042 2Ch. BiSS-C Encoder]
//               AT1K2-EL5042-02 [EL5042 2Ch. BiSS-C Encoder]
//               AT1K2-EL3202-01 [EL3202-0020 2Ch. Ana. Input PT100 (RTD), High Precision, calibrated]
//               AT1K2-EL3202-02 [EL3202-0020 2Ch. Ana. Input PT100 (RTD), High Precision, calibrated]
//               AT1K2-EL3052-E8
//               AT1K2-EL9011
//           Term 73 (EK1122) [EK1122 2 port EtherCAT junction]
//             PAX-DRL-02 (EK1100) [EK1100 EtherCAT Coupler (2A E-Bus)]
//               PAX-EL7047-E01 [EL7047 1Ch. Stepper motor output stage (50V, 5A)]
//               PAX-EL5042-E02 [EL5042 2Ch. BiSS-C Encoder]
//               PAX-EL7047-E03 [EL7047 1Ch. Stepper motor output stage (50V, 5A)]
//               PAX-EL7047-E04 [EL7047 1Ch. Stepper motor output stage (50V, 5A)]
//               PAX-EL5042-E05 [EL5042 2Ch. BiSS-C Encoder]
//               PAX-EL7047-E06 [EL7047 1Ch. Stepper motor output stage (50V, 5A)]
//               PAX-EL2004-E07 [EL2004 4Ch. Dig. Output 24V, 0.5A]
//               PAX-EL7047-E08 [EL7047 1Ch. Stepper motor output stage (50V, 5A)]
//               PAX-EL5042-E09 [EL5042 2Ch. BiSS-C Encoder]
//               PAX-EL7047-E10 [EL7047 1Ch. Stepper motor output stage (50V, 5A)]
//               PAX-EL9410-E11 [EL9410 E-Bus Power Supplier  (Diagnostics)]
//               PAX-EL7047-E12 [EL7047 1Ch. Stepper motor output stage (50V, 5A)]
//               PAX-EL5042-E13 [EL5042 2Ch. BiSS-C Encoder]
//               PAX-EL7047-E14 [EL7047 1Ch. Stepper motor output stage (50V, 5A)]
//               PAX-EL7047-E15 [EL7047 1Ch. Stepper motor output stage (50V, 5A)]
//               PAX-EL5042-E16 [EL5042 2Ch. BiSS-C Encoder]
//               PAX-EL7047-E17 [EL7047 1Ch. Stepper motor output stage (50V, 5A)]
//               PAX-EL9011 [EL9011 End Terminal]
//             K2S18-DRL-02 (EK1100) [EK1100 EtherCAT Coupler (2A E-Bus)]
//               K2S18-DRL-02-E1 (EL7047)
//               K2S18-DRL-02-E2 (EL5042)
//               K2S18-DRL-02-E3 (EL7047)
//               K2S18-DRL-02-E4 (EL7047)
//               K2S18-DRL-02-E5 (EL5042)
//               K2S18-DRL-02-E6 (EL7047) [EL7047 1Ch. Stepper motor output stage (50V, 5A)]
//               K2S18-DRL-02-E7 (EL7047) [EL7047 1Ch. Stepper motor output stage (50V, 5A)]
//               K2S18-DRL-02-E8 (EL5042)
//               K2S18-DRL-02-E9 (EL3202)
//               K2S18-DRL-02-E10 (EL3202)
//               Term 410 (EL9011)
//             K2S18-DRL-03 (EK1100) [EK1100 EtherCAT Coupler (2A E-Bus)]
//               K2S18-DRL-03-E1(EL7047) [EL7047 1Ch. Stepper motor output stage (50V, 5A)]
//               K2S18-DRL-03-E2 (EL5042)
//               K2S18-DRL-03-E3 (EL7047)
//               K2S18-DRL-03-E4 (EL7047) [EL7047 1Ch. Stepper motor output stage (50V, 5A)]
//               K2S18-DRL-03-E5 (EL5042)
//               K2S18-DRL-03-E6 (EL7047)
//               K2S18-DRL-03-E7 (EL7047)
//               K2S18-DRL-03-E8 (EL5112)
//               K2S18-DRL-03-E9 (EL7037)
//               K2S18-DRL-03-E10 (EL7037)
//               K2S18-DRL-03-E11 (EL7037)
//               K2S18-DRL-03-E12 (EL9505)
//               K2S18-DRL-03-E13 (EL1124) [EL1124 4Ch. Dig. Input 5V, 10µs, Sensor Power]
//               K2S18-DRL-03-E14 (EL1124)
//               Term 411 (EL9011) [EL9011 End Terminal]
//           Term 74 (EK1122) [EK1122 2 port EtherCAT junction]
//           Term 75 (EK1110) [EK1110 EtherCAT extension]
//       PLC End Coupler (EK1110)
//     EtherCAT Panel (EK1100) [EK1100 EtherCAT Coupler (2A E-Bus)]
//       EC E1 (EK1122) [EK1122 2 port EtherCAT junction]
//         X1 IM1K1-PPM (EK1100) [EK1100 EtherCAT Coupler (2A E-Bus)]
//           IM1K1-EL7041 [EL7041 1Ch. Stepper motor output stage (50V, 5A)]
//           IM1K1-EL5042 [EL5042 2Ch. BiSS-C Encoder]
//           IM1K1-EL2004 [EL2004 4Ch. Dig. Output 24V, 0.5A]
//           IM1K1-EL3314 [EL3314 4Ch. Ana. Input Thermocouple (TC)]
//           IM1K1-EL3052 [EL3052 2Ch. Ana. Input 4-20mA]
//           IM1K1-EL3062 [EL3062 2Ch. Ana. Input 0-10V]
//           IM1K1-EL4004 [EL4004 4Ch. Ana. Output 0-10V, 12bit]
//           IM1K1-EL9011 [EL9011 End Terminal]
//         X2 IM2K1-PPM (EK1100)
//       EC E2 (EK1122) [EK1122 2 port EtherCAT junction]
//       Term 296 (EL9011) [EL9011 End Terminal]
// variable links:
//   Axes/Axis 25 AT1K2-SOLID-MMS-01 <-> PLC Rail (EtherCAT)/Power (EK1200)/Fiber Coupler (EK1521-0010)/Term 123 (EK1100)/Term 157 (EK1122)/AT1K2-SOLID (EK1100)/AT1K2-EL5042-01
//     Enc/Inputs/In/nComState @bit 1 <-> WcState/InputToggle
//     Enc/Inputs/In/nComState <-> WcState/WcState
//     Enc/Inputs/In/nDataIn1 <-> FB Inputs Channel 1/Position
//     Enc/Inputs/In/nState1 @bit 12 <-> FB Inputs Channel 1/Status/Diag
//     Enc/Inputs/In/nState1 @bit 1 <-> FB Inputs Channel 1/Status/Error
//     Enc/Inputs/In/nState1 @bit 14 <-> FB Inputs Channel 1/Status/Input cycle counter
//     Enc/Inputs/In/nState1 @bit 2 <-> FB Inputs Channel 1/Status/Ready
//     Enc/Inputs/In/nState1 @bit 13 <-> FB Inputs Channel 1/Status/TxPDO State
//     Enc/Inputs/In/nState1 <-> FB Inputs Channel 1/Status/Warning
//   Axes/Axis 25 AT1K2-SOLID-MMS-01 <-> PLC Rail (EtherCAT)/Power (EK1200)/Fiber Coupler (EK1521-0010)/Term 123 (EK1100)/Term 157 (EK1122)/AT1K2-SOLID (EK1100)/AT1K2-EL7047-01
//     Drive/Inputs/In/nState1 @bit 3 <-> STM Status/Status/Error
//     Drive/Inputs/In/nState1 @bit 7 <-> STM Status/Status/Motor stall
//     Drive/Inputs/In/nState1 @bit 5 <-> STM Status/Status/Moving negative
//     Drive/Inputs/In/nState1 @bit 4 <-> STM Status/Status/Moving positive
//     Drive/Inputs/In/nState1 @bit 1 <-> STM Status/Status/Ready
//     Drive/Inputs/In/nState1 <-> STM Status/Status/Ready to enable
//     Drive/Inputs/In/nState1 @bit 6 <-> STM Status/Status/Torque reduced
//     Drive/Inputs/In/nState1 @bit 2 <-> STM Status/Status/Warning
//     Drive/Inputs/In/nState2 @bit 3 <-> STM Status/Status/Digital input 1
//     Drive/Inputs/In/nState2 @bit 4 <-> STM Status/Status/Digital input 2
//     Drive/Inputs/In/nState2 @bit 5 <-> STM Status/Status/Sync error
//     Drive/Inputs/In/nState2 @bit 7 <-> STM Status/Status/TxPDO Toggle
//     Drive/Inputs/In/nState4 @bit 1 <-> WcState/InputToggle
//     Drive/Inputs/In/nState4 <-> WcState/WcState
//     Drive/Outputs/Out/nCtrl1 <-> STM Control/Control/Enable
//     Drive/Outputs/Out/nCtrl1 @bit 2 <-> STM Control/Control/Reduce torque
//     Drive/Outputs/Out/nCtrl1 @bit 1 <-> STM Control/Control/Reset
//     Drive/Outputs/Out/nCtrl2 @bit 3 <-> STM Control/Control/Digital output 1
//     Drive/Outputs/Out/nDataOut2[0] <-> STM Velocity/Velocity
//   Axes/Axis 26 AT1K2-SOLID-MMS-02 <-> PLC Rail (EtherCAT)/Power (EK1200)/Fiber Coupler (EK1521-0010)/Term 123 (EK1100)/Term 157 (EK1122)/AT1K2-SOLID (EK1100)/AT1K2-EL5042-01
//     Enc/Inputs/In/nComState @bit 1 <-> WcState/InputToggle
//     Enc/Inputs/In/nComState <-> WcState/WcState
//     Enc/Inputs/In/nDataIn1 <-> FB Inputs Channel 2/Position
//     Enc/Inputs/In/nState1 @bit 12 <-> FB Inputs Channel 2/Status/Diag
//     Enc/Inputs/In/nState1 @bit 1 <-> FB Inputs Channel 2/Status/Error
//     Enc/Inputs/In/nState1 @bit 14 <-> FB Inputs Channel 2/Status/Input cycle counter
//     Enc/Inputs/In/nState1 @bit 2 <-> FB Inputs Channel 2/Status/Ready
//     Enc/Inputs/In/nState1 @bit 13 <-> FB Inputs Channel 2/Status/TxPDO State
//     Enc/Inputs/In/nState1 <-> FB Inputs Channel 2/Status/Warning
//   Axes/Axis 26 AT1K2-SOLID-MMS-02 <-> PLC Rail (EtherCAT)/Power (EK1200)/Fiber Coupler (EK1521-0010)/Term 123 (EK1100)/Term 157 (EK1122)/AT1K2-SOLID (EK1100)/AT1K2-EL7047-02
//     Drive/Inputs/In/nState1 @bit 3 <-> STM Status/Status/Error
//     Drive/Inputs/In/nState1 @bit 7 <-> STM Status/Status/Motor stall
//     Drive/Inputs/In/nState1 @bit 5 <-> STM Status/Status/Moving negative
//     Drive/Inputs/In/nState1 @bit 4 <-> STM Status/Status/Moving positive
//     Drive/Inputs/In/nState1 @bit 1 <-> STM Status/Status/Ready
//     Drive/Inputs/In/nState1 <-> STM Status/Status/Ready to enable
//     Drive/Inputs/In/nState1 @bit 6 <-> STM Status/Status/Torque reduced
//     Drive/Inputs/In/nState1 @bit 2 <-> STM Status/Status/Warning
//     Drive/Inputs/In/nState2 @bit 3 <-> STM Status/Status/Digital input 1
//     Drive/Inputs/In/nState2 @bit 4 <-> STM Status/Status/Digital input 2
//     Drive/Inputs/In/nState2 @bit 5 <-> STM Status/Status/Sync error
//     Drive/Inputs/In/nState2 @bit 7 <-> STM Status/Status/TxPDO Toggle
//     Drive/Inputs/In/nState4 @bit 1 <-> WcState/InputToggle
//     Drive/Inputs/In/nState4 <-> WcState/WcState
//     Drive/Outputs/Out/nCtrl1 <-> STM Control/Control/Enable
//     Drive/Outputs/Out/nCtrl1 @bit 2 <-> STM Control/Control/Reduce torque
//     Drive/Outputs/Out/nCtrl1 @bit 1 <-> STM Control/Control/Reset
//     Drive/Outputs/Out/nCtrl2 @bit 3 <-> STM Control/Control/Digital output 1
//     Drive/Outputs/Out/nDataOut2[0] <-> STM Velocity/Velocity
//   Axes/Axis 27 AT1K2-SOLID-MMS-03 <-> PLC Rail (EtherCAT)/Power (EK1200)/Fiber Coupler (EK1521-0010)/Term 123 (EK1100)/Term 157 (EK1122)/AT1K2-SOLID (EK1100)/AT1K2-EL5042-02
//     Enc/Inputs/In/nComState @bit 1 <-> WcState/InputToggle
//     Enc/Inputs/In/nComState <-> WcState/WcState
//     Enc/Inputs/In/nDataIn1 <-> FB Inputs Channel 1/Position
//     Enc/Inputs/In/nState1 @bit 12 <-> FB Inputs Channel 1/Status/Diag
//     Enc/Inputs/In/nState1 @bit 1 <-> FB Inputs Channel 1/Status/Error
//     Enc/Inputs/In/nState1 @bit 14 <-> FB Inputs Channel 1/Status/Input cycle counter
//     Enc/Inputs/In/nState1 @bit 2 <-> FB Inputs Channel 1/Status/Ready
//     Enc/Inputs/In/nState1 @bit 13 <-> FB Inputs Channel 1/Status/TxPDO State
//     Enc/Inputs/In/nState1 <-> FB Inputs Channel 1/Status/Warning
//   Axes/Axis 27 AT1K2-SOLID-MMS-03 <-> PLC Rail (EtherCAT)/Power (EK1200)/Fiber Coupler (EK1521-0010)/Term 123 (EK1100)/Term 157 (EK1122)/AT1K2-SOLID (EK1100)/AT1K2-EL7047-03
//     Drive/Inputs/In/nState1 @bit 3 <-> STM Status/Status/Error
//     Drive/Inputs/In/nState1 @bit 7 <-> STM Status/Status/Motor stall
//     Drive/Inputs/In/nState1 @bit 5 <-> STM Status/Status/Moving negative
//     Drive/Inputs/In/nState1 @bit 4 <-> STM Status/Status/Moving positive
//     Drive/Inputs/In/nState1 @bit 1 <-> STM Status/Status/Ready
//     Drive/Inputs/In/nState1 <-> STM Status/Status/Ready to enable
//     Drive/Inputs/In/nState1 @bit 6 <-> STM Status/Status/Torque reduced
//     Drive/Inputs/In/nState1 @bit 2 <-> STM Status/Status/Warning
//     Drive/Inputs/In/nState2 @bit 3 <-> STM Status/Status/Digital input 1
//     Drive/Inputs/In/nState2 @bit 4 <-> STM Status/Status/Digital input 2
//     Drive/Inputs/In/nState2 @bit 5 <-> STM Status/Status/Sync error
//     Drive/Inputs/In/nState2 @bit 7 <-> STM Status/Status/TxPDO Toggle
//     Drive/Inputs/In/nState4 @bit 1 <-> WcState/InputToggle
//     Drive/Inputs/In/nState4 <-> WcState/WcState
//     Drive/Outputs/Out/nCtrl1 <-> STM Control/Control/Enable
//     Drive/Outputs/Out/nCtrl1 @bit 2 <-> STM Control/Control/Reduce torque
//     Drive/Outputs/Out/nCtrl1 @bit 1 <-> STM Control/Control/Reset
//     Drive/Outputs/Out/nCtrl2 @bit 3 <-> STM Control/Control/Digital output 1
//     Drive/Outputs/Out/nDataOut2[0] <-> STM Velocity/Velocity
//   (this object) <-> PLC Rail (EtherCAT)/EtherCAT Panel (EK1100)/EC E1 (EK1122)/X1 IM1K1-PPM (EK1100)/IM1K1-EL5042
//     Enc/Inputs/In/nComState @bit 1 <-> WcState/InputToggle
//     Enc/Inputs/In/nComState <-> WcState/WcState
//     Enc/Inputs/In/nDataIn1 <-> FB Inputs Channel 1/Position
//     Enc/Inputs/In/nState1 @bit 12 <-> FB Inputs Channel 1/Status/Diag
//     Enc/Inputs/In/nState1 @bit 1 <-> FB Inputs Channel 1/Status/Error
//     Enc/Inputs/In/nState1 @bit 14 <-> FB Inputs Channel 1/Status/Input cycle counter
//     Enc/Inputs/In/nState1 @bit 2 <-> FB Inputs Channel 1/Status/Ready
//     Enc/Inputs/In/nState1 @bit 13 <-> FB Inputs Channel 1/Status/TxPDO State
//     Enc/Inputs/In/nState1 <-> FB Inputs Channel 1/Status/Warning
//   (this object) <-> PLC Rail (EtherCAT)/EtherCAT Panel (EK1100)/EC E1 (EK1122)/X1 IM1K1-PPM (EK1100)/IM1K1-EL7041
//     Drive/Inputs/In/nState1 @bit 3 <-> STM Status/Status/Error
//     Drive/Inputs/In/nState1 @bit 5 <-> STM Status/Status/Moving negative
//     Drive/Inputs/In/nState1 @bit 4 <-> STM Status/Status/Moving positive
//     Drive/Inputs/In/nState1 @bit 1 <-> STM Status/Status/Ready
//     Drive/Inputs/In/nState1 <-> STM Status/Status/Ready to enable
//     Drive/Inputs/In/nState1 @bit 6 <-> STM Status/Status/Torque reduced
//     Drive/Inputs/In/nState1 @bit 2 <-> STM Status/Status/Warning
//     Drive/Inputs/In/nState2 @bit 3 <-> STM Status/Status/Digital input 1
//     Drive/Inputs/In/nState2 @bit 4 <-> STM Status/Status/Digital input 2
//     Drive/Inputs/In/nState2 @bit 5 <-> STM Status/Status/Sync error
//     Drive/Inputs/In/nState2 @bit 7 <-> STM Status/Status/TxPDO Toggle
//     Drive/Inputs/In/nState4 @bit 1 <-> WcState/InputToggle
//     Drive/Inputs/In/nState4 <-> WcState/WcState
//     Drive/Outputs/Out/nCtrl1 <-> STM Control/Control/Enable
//     Drive/Outputs/Out/nCtrl1 @bit 2 <-> STM Control/Control/Reduce torque
//     Drive/Outputs/Out/nCtrl1 @bit 1 <-> STM Control/Control/Reset
//     Drive/Outputs/Out/nDataOut2[0] <-> STM Velocity/Velocity
//   (this object) <-> PLC Rail (EtherCAT)/EtherCAT Panel (EK1100)/EC E1 (EK1122)/X2 IM2K1-PPM (EK1100)/IM2K1-EL5042
//     Enc/Inputs/In/nComState @bit 1 <-> WcState/InputToggle
//     Enc/Inputs/In/nComState <-> WcState/WcState
//     Enc/Inputs/In/nDataIn1 <-> FB Inputs Channel 1/Position
//     Enc/Inputs/In/nState1 @bit 12 <-> FB Inputs Channel 1/Status/Diag
//     Enc/Inputs/In/nState1 @bit 1 <-> FB Inputs Channel 1/Status/Error
//     Enc/Inputs/In/nState1 @bit 14 <-> FB Inputs Channel 1/Status/Input cycle counter
//     Enc/Inputs/In/nState1 @bit 2 <-> FB Inputs Channel 1/Status/Ready
//     Enc/Inputs/In/nState1 @bit 13 <-> FB Inputs Channel 1/Status/TxPDO State
//     Enc/Inputs/In/nState1 <-> FB Inputs Channel 1/Status/Warning
//   (this object) <-> PLC Rail (EtherCAT)/EtherCAT Panel (EK1100)/EC E1 (EK1122)/X2 IM2K1-PPM (EK1100)/IM2K1-EL7041
//     Drive/Inputs/In/nState1 @bit 3 <-> STM Status/Status/Error
//     Drive/Inputs/In/nState1 @bit 5 <-> STM Status/Status/Moving negative
//     Drive/Inputs/In/nState1 @bit 4 <-> STM Status/Status/Moving positive
//     Drive/Inputs/In/nState1 @bit 1 <-> STM Status/Status/Ready
//     Drive/Inputs/In/nState1 <-> STM Status/Status/Ready to enable
//     Drive/Inputs/In/nState1 @bit 6 <-> STM Status/Status/Torque reduced
//     Drive/Inputs/In/nState1 @bit 2 <-> STM Status/Status/Warning
//     Drive/Inputs/In/nState2 @bit 3 <-> STM Status/Status/Digital input 1
//     Drive/Inputs/In/nState2 @bit 4 <-> STM Status/Status/Digital input 2
//     Drive/Inputs/In/nState2 @bit 5 <-> STM Status/Status/Sync error
//     Drive/Inputs/In/nState2 @bit 7 <-> STM Status/Status/TxPDO Toggle
//     Drive/Inputs/In/nState4 @bit 1 <-> WcState/InputToggle
//     Drive/Inputs/In/nState4 <-> WcState/WcState
//     Drive/Outputs/Out/nCtrl1 <-> STM Control/Control/Enable
//     Drive/Outputs/Out/nCtrl1 @bit 2 <-> STM Control/Control/Reduce torque
//     Drive/Outputs/Out/nCtrl1 @bit 1 <-> STM Control/Control/Reset
//     Drive/Outputs/Out/nDataOut2[0] <-> STM Velocity/Velocity
//   (this object) <-> PLC Rail (EtherCAT)/Power (EK1200)/Fiber Coupler (EK1521-0010)/Term 34 (EK1501-0010)/Term 39 (EK1122)/IM1K2-PPM (EK1100)/IM1K2-EL5042-E2
//     Enc/Inputs/In/nComState @bit 1 <-> WcState/InputToggle
//     Enc/Inputs/In/nComState <-> WcState/WcState
//     Enc/Inputs/In/nDataIn1 <-> FB Inputs Channel 1/Position
//     Enc/Inputs/In/nState1 @bit 12 <-> FB Inputs Channel 1/Status/Diag
//     Enc/Inputs/In/nState1 @bit 1 <-> FB Inputs Channel 1/Status/Error
//     Enc/Inputs/In/nState1 @bit 14 <-> FB Inputs Channel 1/Status/Input cycle counter
//     Enc/Inputs/In/nState1 @bit 2 <-> FB Inputs Channel 1/Status/Ready
//     Enc/Inputs/In/nState1 @bit 13 <-> FB Inputs Channel 1/Status/TxPDO State
//     Enc/Inputs/In/nState1 <-> FB Inputs Channel 1/Status/Warning
//   (this object) <-> PLC Rail (EtherCAT)/Power (EK1200)/Fiber Coupler (EK1521-0010)/Term 34 (EK1501-0010)/Term 39 (EK1122)/IM1K2-PPM (EK1100)/IM1K2-EL7041-E1
//     Drive/Inputs/In/nState1 @bit 3 <-> STM Status/Status/Error
//     Drive/Inputs/In/nState1 @bit 5 <-> STM Status/Status/Moving negative
//     Drive/Inputs/In/nState1 @bit 4 <-> STM Status/Status/Moving positive
//     Drive/Inputs/In/nState1 @bit 1 <-> STM Status/Status/Ready
//     Drive/Inputs/In/nState1 <-> STM Status/Status/Ready to enable
//     Drive/Inputs/In/nState1 @bit 6 <-> STM Status/Status/Torque reduced
//     Drive/Inputs/In/nState1 @bit 2 <-> STM Status/Status/Warning
//     Drive/Inputs/In/nState2 @bit 3 <-> STM Status/Status/Digital input 1
//     Drive/Inputs/In/nState2 @bit 4 <-> STM Status/Status/Digital input 2
//     Drive/Inputs/In/nState2 @bit 5 <-> STM Status/Status/Sync error
//     Drive/Inputs/In/nState2 @bit 7 <-> STM Status/Status/TxPDO Toggle
//     Drive/Inputs/In/nState4 @bit 1 <-> WcState/InputToggle
//     Drive/Inputs/In/nState4 <-> WcState/WcState
//     Drive/Outputs/Out/nCtrl1 <-> STM Control/Control/Enable
//     Drive/Outputs/Out/nCtrl1 @bit 2 <-> STM Control/Control/Reduce torque
//     Drive/Outputs/Out/nCtrl1 @bit 1 <-> STM Control/Control/Reset
//     Drive/Outputs/Out/nDataOut2[0] <-> STM Velocity/Velocity
//   (this object) <-> PLC Rail (EtherCAT)/Power (EK1200)/Fiber Coupler (EK1521-0010)/Term 123 (EK1100)/Term 124 (EK1122)/TM1K2-K2A (EK1100)/TM1K2-EL5042-E3
//     Enc/Inputs/In/nComState @bit 1 <-> WcState/InputToggle
//     Enc/Inputs/In/nComState <-> WcState/WcState
//     Enc/Inputs/In/nDataIn1 <-> FB Inputs Channel 1/Position
//     Enc/Inputs/In/nDataIn1 <-> FB Inputs Channel 2/Position
//     Enc/Inputs/In/nState1 @bit 12 <-> FB Inputs Channel 1/Status/Diag
//     Enc/Inputs/In/nState1 @bit 12 <-> FB Inputs Channel 2/Status/Diag
//     Enc/Inputs/In/nState1 @bit 1 <-> FB Inputs Channel 1/Status/Error
//     Enc/Inputs/In/nState1 @bit 1 <-> FB Inputs Channel 2/Status/Error
//     Enc/Inputs/In/nState1 @bit 14 <-> FB Inputs Channel 1/Status/Input cycle counter
//     Enc/Inputs/In/nState1 @bit 14 <-> FB Inputs Channel 2/Status/Input cycle counter
//     Enc/Inputs/In/nState1 @bit 2 <-> FB Inputs Channel 1/Status/Ready
//     Enc/Inputs/In/nState1 @bit 2 <-> FB Inputs Channel 2/Status/Ready
//     Enc/Inputs/In/nState1 @bit 13 <-> FB Inputs Channel 1/Status/TxPDO State
//     Enc/Inputs/In/nState1 @bit 13 <-> FB Inputs Channel 2/Status/TxPDO State
//     Enc/Inputs/In/nState1 <-> FB Inputs Channel 1/Status/Warning
//     Enc/Inputs/In/nState1 <-> FB Inputs Channel 2/Status/Warning
//   (this object) <-> PLC Rail (EtherCAT)/Power (EK1200)/Fiber Coupler (EK1521-0010)/Term 123 (EK1100)/Term 124 (EK1122)/TM1K2-K2A (EK1100)/TM1K2-EL7041-E1
//     Drive/Inputs/In/nState1 @bit 3 <-> STM Status/Status/Error
//     Drive/Inputs/In/nState1 @bit 5 <-> STM Status/Status/Moving negative
//     Drive/Inputs/In/nState1 @bit 4 <-> STM Status/Status/Moving positive
//     Drive/Inputs/In/nState1 @bit 1 <-> STM Status/Status/Ready
//     Drive/Inputs/In/nState1 <-> STM Status/Status/Ready to enable
//     Drive/Inputs/In/nState1 @bit 6 <-> STM Status/Status/Torque reduced
//     Drive/Inputs/In/nState1 @bit 2 <-> STM Status/Status/Warning
//     Drive/Inputs/In/nState2 @bit 3 <-> STM Status/Status/Digital input 1
//     Drive/Inputs/In/nState2 @bit 4 <-> STM Status/Status/Digital input 2
//     Drive/Inputs/In/nState2 @bit 5 <-> STM Status/Status/Sync error
//     Drive/Inputs/In/nState2 @bit 7 <-> STM Status/Status/TxPDO Toggle
//     Drive/Inputs/In/nState4 @bit 1 <-> WcState/InputToggle
//     Drive/Inputs/In/nState4 <-> WcState/WcState
//     Drive/Outputs/Out/nCtrl1 <-> STM Control/Control/Enable
//     Drive/Outputs/Out/nCtrl1 @bit 2 <-> STM Control/Control/Reduce torque
//     Drive/Outputs/Out/nCtrl1 @bit 1 <-> STM Control/Control/Reset
//     Drive/Outputs/Out/nDataOut2[0] <-> STM Velocity/Velocity
//   (this object) <-> PLC Rail (EtherCAT)/Power (EK1200)/Fiber Coupler (EK1521-0010)/Term 123 (EK1100)/Term 124 (EK1122)/TM1K2-K2A (EK1100)/TM1K2-EL7041-E2
//     Drive/Inputs/In/nState1 @bit 3 <-> STM Status/Status/Error
//     Drive/Inputs/In/nState1 @bit 5 <-> STM Status/Status/Moving negative
//     Drive/Inputs/In/nState1 @bit 4 <-> STM Status/Status/Moving positive
//     Drive/Inputs/In/nState1 @bit 1 <-> STM Status/Status/Ready
//     Drive/Inputs/In/nState1 <-> STM Status/Status/Ready to enable
//     Drive/Inputs/In/nState1 @bit 6 <-> STM Status/Status/Torque reduced
//     Drive/Inputs/In/nState1 @bit 2 <-> STM Status/Status/Warning
//     Drive/Inputs/In/nState2 @bit 3 <-> STM Status/Status/Digital input 1
//     Drive/Inputs/In/nState2 @bit 4 <-> STM Status/Status/Digital input 2
//     Drive/Inputs/In/nState2 @bit 5 <-> STM Status/Status/Sync error
//     Drive/Inputs/In/nState2 @bit 7 <-> STM Status/Status/TxPDO Toggle
//     Drive/Inputs/In/nState4 @bit 1 <-> WcState/InputToggle
//     Drive/Inputs/In/nState4 <-> WcState/WcState
//     Drive/Outputs/Out/nCtrl1 <-> STM Control/Control/Enable
//     Drive/Outputs/Out/nCtrl1 @bit 2 <-> STM Control/Control/Reduce torque
//     Drive/Outputs/Out/nCtrl1 @bit 1 <-> STM Control/Control/Reset
//     Drive/Outputs/Out/nDataOut2[0] <-> STM Velocity/Velocity
//   (this object) <-> PLC Rail (EtherCAT)/Power (EK1200)/Fiber Coupler (EK1521-0010)/Term 34 (EK1501-0010)/Term 49 (EK1122)/IM2K2-PPM (EK1100)/IM2K2-EL5042-E2
//     Enc/Inputs/In/nComState @bit 1 <-> WcState/InputToggle
//     Enc/Inputs/In/nComState <-> WcState/WcState
//     Enc/Inputs/In/nDataIn1 <-> FB Inputs Channel 1/Position
//     Enc/Inputs/In/nState1 @bit 12 <-> FB Inputs Channel 1/Status/Diag
//     Enc/Inputs/In/nState1 @bit 1 <-> FB Inputs Channel 1/Status/Error
//     Enc/Inputs/In/nState1 @bit 14 <-> FB Inputs Channel 1/Status/Input cycle counter
//     Enc/Inputs/In/nState1 @bit 2 <-> FB Inputs Channel 1/Status/Ready
//     Enc/Inputs/In/nState1 @bit 13 <-> FB Inputs Channel 1/Status/TxPDO State
//     Enc/Inputs/In/nState1 <-> FB Inputs Channel 1/Status/Warning
//   (this object) <-> PLC Rail (EtherCAT)/Power (EK1200)/Fiber Coupler (EK1521-0010)/Term 34 (EK1501-0010)/Term 49 (EK1122)/IM2K2-PPM (EK1100)/IM2K2-EL7041-E1
//     Drive/Inputs/In/nState1 @bit 3 <-> STM Status/Status/Error
//     Drive/Inputs/In/nState1 @bit 5 <-> STM Status/Status/Moving negative
//     Drive/Inputs/In/nState1 @bit 4 <-> STM Status/Status/Moving positive
//     Drive/Inputs/In/nState1 @bit 1 <-> STM Status/Status/Ready
//     Drive/Inputs/In/nState1 <-> STM Status/Status/Ready to enable
//     Drive/Inputs/In/nState1 @bit 6 <-> STM Status/Status/Torque reduced
//     Drive/Inputs/In/nState1 @bit 2 <-> STM Status/Status/Warning
//     Drive/Inputs/In/nState2 @bit 3 <-> STM Status/Status/Digital input 1
//     Drive/Inputs/In/nState2 @bit 4 <-> STM Status/Status/Digital input 2
//     Drive/Inputs/In/nState2 @bit 5 <-> STM Status/Status/Sync error
//     Drive/Inputs/In/nState2 @bit 7 <-> STM Status/Status/TxPDO Toggle
//     Drive/Inputs/In/nState4 @bit 1 <-> WcState/InputToggle
//     Drive/Inputs/In/nState4 <-> WcState/WcState
//     Drive/Outputs/Out/nCtrl1 <-> STM Control/Control/Enable
//     Drive/Outputs/Out/nCtrl1 @bit 2 <-> STM Control/Control/Reduce torque
//     Drive/Outputs/Out/nCtrl1 @bit 1 <-> STM Control/Control/Reset
//     Drive/Outputs/Out/nDataOut2[0] <-> STM Velocity/Velocity
//   (this object) <-> PLC Rail (EtherCAT)/Power (EK1200)/Fiber Coupler (EK1521-0010)/Term 34 (EK1501-0010)/Term 50 (EK1122)/IM3K2-PPM (EK1100)/IM3K2-EL5042-E2
//     Enc/Inputs/In/nComState @bit 1 <-> WcState/InputToggle
//     Enc/Inputs/In/nComState <-> WcState/WcState
//     Enc/Inputs/In/nDataIn1 <-> FB Inputs Channel 1/Position
//     Enc/Inputs/In/nState1 @bit 12 <-> FB Inputs Channel 1/Status/Diag
//     Enc/Inputs/In/nState1 @bit 1 <-> FB Inputs Channel 1/Status/Error
//     Enc/Inputs/In/nState1 @bit 14 <-> FB Inputs Channel 1/Status/Input cycle counter
//     Enc/Inputs/In/nState1 @bit 2 <-> FB Inputs Channel 1/Status/Ready
//     Enc/Inputs/In/nState1 @bit 13 <-> FB Inputs Channel 1/Status/TxPDO State
//     Enc/Inputs/In/nState1 <-> FB Inputs Channel 1/Status/Warning
//   (this object) <-> PLC Rail (EtherCAT)/Power (EK1200)/Fiber Coupler (EK1521-0010)/Term 34 (EK1501-0010)/Term 50 (EK1122)/IM3K2-PPM (EK1100)/IM3K2-EL7041-E1
//     Drive/Inputs/In/nState1 @bit 3 <-> STM Status/Status/Error
//     Drive/Inputs/In/nState1 @bit 5 <-> STM Status/Status/Moving negative
//     Drive/Inputs/In/nState1 @bit 4 <-> STM Status/Status/Moving positive
//     Drive/Inputs/In/nState1 @bit 1 <-> STM Status/Status/Ready
//     Drive/Inputs/In/nState1 <-> STM Status/Status/Ready to enable
//     Drive/Inputs/In/nState1 @bit 6 <-> STM Status/Status/Torque reduced
//     Drive/Inputs/In/nState1 @bit 2 <-> STM Status/Status/Warning
//     Drive/Inputs/In/nState2 @bit 3 <-> STM Status/Status/Digital input 1
//     Drive/Inputs/In/nState2 @bit 4 <-> STM Status/Status/Digital input 2
//     Drive/Inputs/In/nState2 @bit 5 <-> STM Status/Status/Sync error
//     Drive/Inputs/In/nState2 @bit 7 <-> STM Status/Status/TxPDO Toggle
//     Drive/Inputs/In/nState4 @bit 1 <-> WcState/InputToggle
//     Drive/Inputs/In/nState4 <-> WcState/WcState
//     Drive/Outputs/Out/nCtrl1 <-> STM Control/Control/Enable
//     Drive/Outputs/Out/nCtrl1 @bit 2 <-> STM Control/Control/Reduce torque
//     Drive/Outputs/Out/nCtrl1 @bit 1 <-> STM Control/Control/Reset
//     Drive/Outputs/Out/nDataOut2[0] <-> STM Velocity/Velocity
//   (this object) <-> PLC Rail (EtherCAT)/Power (EK1200)/Fiber Coupler (EK1521-0010)/Term 34 (EK1501-0010)/Term 50 (EK1122)/IM4K2-PPM (EK1100)/IM4K2-EL5042-E2
//     Enc/Inputs/In/nComState @bit 1 <-> WcState/InputToggle
//     Enc/Inputs/In/nComState <-> WcState/WcState
//     Enc/Inputs/In/nDataIn1 <-> FB Inputs Channel 1/Position
//     Enc/Inputs/In/nState1 @bit 12 <-> FB Inputs Channel 1/Status/Diag
//     Enc/Inputs/In/nState1 @bit 1 <-> FB Inputs Channel 1/Status/Error
//     Enc/Inputs/In/nState1 @bit 14 <-> FB Inputs Channel 1/Status/Input cycle counter
//     Enc/Inputs/In/nState1 @bit 2 <-> FB Inputs Channel 1/Status/Ready
//     Enc/Inputs/In/nState1 @bit 13 <-> FB Inputs Channel 1/Status/TxPDO State
//     Enc/Inputs/In/nState1 <-> FB Inputs Channel 1/Status/Warning
//   (this object) <-> PLC Rail (EtherCAT)/Power (EK1200)/Fiber Coupler (EK1521-0010)/Term 34 (EK1501-0010)/Term 50 (EK1122)/IM4K2-PPM (EK1100)/IM4K2-EL7041-E1
//     Drive/Inputs/In/nState1 @bit 3 <-> STM Status/Status/Error
//     Drive/Inputs/In/nState1 @bit 5 <-> STM Status/Status/Moving negative
//     Drive/Inputs/In/nState1 @bit 4 <-> STM Status/Status/Moving positive
//     Drive/Inputs/In/nState1 @bit 1 <-> STM Status/Status/Ready
//     Drive/Inputs/In/nState1 <-> STM Status/Status/Ready to enable
//     Drive/Inputs/In/nState1 @bit 6 <-> STM Status/Status/Torque reduced
//     Drive/Inputs/In/nState1 @bit 2 <-> STM Status/Status/Warning
//     Drive/Inputs/In/nState2 @bit 3 <-> STM Status/Status/Digital input 1
//     Drive/Inputs/In/nState2 @bit 4 <-> STM Status/Status/Digital input 2
//     Drive/Inputs/In/nState2 @bit 5 <-> STM Status/Status/Sync error
//     Drive/Inputs/In/nState2 @bit 7 <-> STM Status/Status/TxPDO Toggle
//     Drive/Inputs/In/nState4 @bit 1 <-> WcState/InputToggle
//     Drive/Inputs/In/nState4 <-> WcState/WcState
//     Drive/Outputs/Out/nCtrl1 <-> STM Control/Control/Enable
//     Drive/Outputs/Out/nCtrl1 @bit 2 <-> STM Control/Control/Reduce torque
//     Drive/Outputs/Out/nCtrl1 @bit 1 <-> STM Control/Control/Reset
//     Drive/Outputs/Out/nDataOut2[0] <-> STM Velocity/Velocity
//   (this object) <-> PLC Rail (EtherCAT)/Power (EK1200)/Fiber Coupler (EK1521-0010)/Term 123 (EK1100)/Term 140 (EK1122)/IM5K2-PPM (EK1100)/IM5K2-EL5042-E2
//     Enc/Inputs/In/nComState @bit 1 <-> WcState/InputToggle
//     Enc/Inputs/In/nComState <-> WcState/WcState
//     Enc/Inputs/In/nDataIn1 <-> FB Inputs Channel 1/Position
//     Enc/Inputs/In/nState1 @bit 12 <-> FB Inputs Channel 1/Status/Diag
//     Enc/Inputs/In/nState1 @bit 1 <-> FB Inputs Channel 1/Status/Error
//     Enc/Inputs/In/nState1 @bit 14 <-> FB Inputs Channel 1/Status/Input cycle counter
//     Enc/Inputs/In/nState1 @bit 2 <-> FB Inputs Channel 1/Status/Ready
//     Enc/Inputs/In/nState1 @bit 13 <-> FB Inputs Channel 1/Status/TxPDO State
//     Enc/Inputs/In/nState1 <-> FB Inputs Channel 1/Status/Warning
//   (this object) <-> PLC Rail (EtherCAT)/Power (EK1200)/Fiber Coupler (EK1521-0010)/Term 123 (EK1100)/Term 140 (EK1122)/IM5K2-PPM (EK1100)/IM5K2-EL7041-E1
//     Drive/Inputs/In/nState1 @bit 3 <-> STM Status/Status/Error
//     Drive/Inputs/In/nState1 @bit 5 <-> STM Status/Status/Moving negative
//     Drive/Inputs/In/nState1 @bit 4 <-> STM Status/Status/Moving positive
//     Drive/Inputs/In/nState1 @bit 1 <-> STM Status/Status/Ready
//     Drive/Inputs/In/nState1 <-> STM Status/Status/Ready to enable
//     Drive/Inputs/In/nState1 @bit 6 <-> STM Status/Status/Torque reduced
//     Drive/Inputs/In/nState1 @bit 2 <-> STM Status/Status/Warning
//     Drive/Inputs/In/nState2 @bit 3 <-> STM Status/Status/Digital input 1
//     Drive/Inputs/In/nState2 @bit 4 <-> STM Status/Status/Digital input 2
//     Drive/Inputs/In/nState2 @bit 5 <-> STM Status/Status/Sync error
//     Drive/Inputs/In/nState2 @bit 7 <-> STM Status/Status/TxPDO Toggle
//     Drive/Inputs/In/nState4 @bit 1 <-> WcState/InputToggle
//     Drive/Inputs/In/nState4 <-> WcState/WcState
//     Drive/Outputs/Out/nCtrl1 <-> STM Control/Control/Enable
//     Drive/Outputs/Out/nCtrl1 @bit 2 <-> STM Control/Control/Reduce torque
//     Drive/Outputs/Out/nCtrl1 @bit 1 <-> STM Control/Control/Reset
//     Drive/Outputs/Out/nDataOut2[0] <-> STM Velocity/Velocity
//   (this object) <-> PLC Rail (EtherCAT)/Power (EK1200)/Fiber Coupler (EK1521-0010)/Term 34 (EK1501-0010)/Term 39 (EK1122)/AL1K2-L2SI (EK1100)/AL1K2-EL5042-E2
//     Enc/Inputs/In/nComState @bit 1 <-> WcState/InputToggle
//     Enc/Inputs/In/nComState <-> WcState/WcState
//     Enc/Inputs/In/nDataIn1 <-> FB Inputs Channel 1/Position
//     Enc/Inputs/In/nState1 @bit 12 <-> FB Inputs Channel 1/Status/Diag
//     Enc/Inputs/In/nState1 @bit 1 <-> FB Inputs Channel 1/Status/Error
//     Enc/Inputs/In/nState1 @bit 14 <-> FB Inputs Channel 1/Status/Input cycle counter
//     Enc/Inputs/In/nState1 @bit 2 <-> FB Inputs Channel 1/Status/Ready
//     Enc/Inputs/In/nState1 @bit 13 <-> FB Inputs Channel 1/Status/TxPDO State
//     Enc/Inputs/In/nState1 <-> FB Inputs Channel 1/Status/Warning
//   (this object) <-> PLC Rail (EtherCAT)/Power (EK1200)/Fiber Coupler (EK1521-0010)/Term 34 (EK1501-0010)/Term 39 (EK1122)/AL1K2-L2SI (EK1100)/AL1K2-EL7041-E1
//     Drive/Inputs/In/nState1 @bit 3 <-> STM Status/Status/Error
//     Drive/Inputs/In/nState1 @bit 5 <-> STM Status/Status/Moving negative
//     Drive/Inputs/In/nState1 @bit 4 <-> STM Status/Status/Moving positive
//     Drive/Inputs/In/nState1 @bit 1 <-> STM Status/Status/Ready
//     Drive/Inputs/In/nState1 <-> STM Status/Status/Ready to enable
//     Drive/Inputs/In/nState1 @bit 6 <-> STM Status/Status/Torque reduced
//     Drive/Inputs/In/nState1 @bit 2 <-> STM Status/Status/Warning
//     Drive/Inputs/In/nState2 @bit 3 <-> STM Status/Status/Digital input 1
//     Drive/Inputs/In/nState2 @bit 4 <-> STM Status/Status/Digital input 2
//     Drive/Inputs/In/nState2 @bit 5 <-> STM Status/Status/Sync error
//     Drive/Inputs/In/nState2 @bit 7 <-> STM Status/Status/TxPDO Toggle
//     Drive/Inputs/In/nState4 @bit 1 <-> WcState/InputToggle
//     Drive/Inputs/In/nState4 <-> WcState/WcState
//     Drive/Outputs/Out/nCtrl1 <-> STM Control/Control/Enable
//     Drive/Outputs/Out/nCtrl1 @bit 2 <-> STM Control/Control/Reduce torque
//     Drive/Outputs/Out/nCtrl1 @bit 1 <-> STM Control/Control/Reset
//     Drive/Outputs/Out/nDataOut2[0] <-> STM Velocity/Velocity
//   (this object) <-> PLC Rail (EtherCAT)/Power (EK1200)/Fiber Coupler (EK1521-0010)/Term 123 (EK1100)/Term 131 (EK1122)/LI2K2-K2A_OUT  (EK1100)/LI2K2-EL5042-E3
//     Enc/Inputs/In/nComState @bit 1 <-> WcState/InputToggle
//     Enc/Inputs/In/nComState <-> WcState/WcState
//     Enc/Inputs/In/nDataIn1 <-> FB Inputs Channel 1/Position
//     Enc/Inputs/In/nState1 @bit 12 <-> FB Inputs Channel 1/Status/Diag
//     Enc/Inputs/In/nState1 @bit 1 <-> FB Inputs Channel 1/Status/Error
//     Enc/Inputs/In/nState1 @bit 14 <-> FB Inputs Channel 1/Status/Input cycle counter
//     Enc/Inputs/In/nState1 @bit 2 <-> FB Inputs Channel 1/Status/Ready
//     Enc/Inputs/In/nState1 @bit 13 <-> FB Inputs Channel 1/Status/TxPDO State
//     Enc/Inputs/In/nState1 <-> FB Inputs Channel 1/Status/Warning
//   (this object) <-> PLC Rail (EtherCAT)/Power (EK1200)/Fiber Coupler (EK1521-0010)/Term 123 (EK1100)/Term 131 (EK1122)/LI2K2-K2A_OUT  (EK1100)/LI2K2-EL7041-E1
//     Drive/Inputs/In/nState1 @bit 3 <-> STM Status/Status/Error
//     Drive/Inputs/In/nState1 @bit 5 <-> STM Status/Status/Moving negative
//     Drive/Inputs/In/nState1 @bit 4 <-> STM Status/Status/Moving positive
//     Drive/Inputs/In/nState1 @bit 1 <-> STM Status/Status/Ready
//     Drive/Inputs/In/nState1 <-> STM Status/Status/Ready to enable
//     Drive/Inputs/In/nState1 @bit 6 <-> STM Status/Status/Torque reduced
//     Drive/Inputs/In/nState1 @bit 2 <-> STM Status/Status/Warning
//     Drive/Inputs/In/nState2 @bit 3 <-> STM Status/Status/Digital input 1
//     Drive/Inputs/In/nState2 @bit 4 <-> STM Status/Status/Digital input 2
//     Drive/Inputs/In/nState2 @bit 5 <-> STM Status/Status/Sync error
//     Drive/Inputs/In/nState2 @bit 7 <-> STM Status/Status/TxPDO Toggle
//     Drive/Inputs/In/nState4 @bit 1 <-> WcState/InputToggle
//     Drive/Inputs/In/nState4 <-> WcState/WcState
//     Drive/Outputs/Out/nCtrl1 <-> STM Control/Control/Enable
//     Drive/Outputs/Out/nCtrl1 @bit 2 <-> STM Control/Control/Reduce torque
//     Drive/Outputs/Out/nCtrl1 @bit 1 <-> STM Control/Control/Reset
//     Drive/Outputs/Out/nDataOut2[0] <-> STM Velocity/Velocity
//   (this object) <-> PLC Rail (EtherCAT)/Power (EK1200)/Fiber Coupler (EK1521-0010)/Term 123 (EK1100)/Term 131 (EK1122)/PF1K2-WFS (EK1100)/PF1K2-EL5042-E3
//     Enc/Inputs/In/nComState @bit 1 <-> WcState/InputToggle
//     Enc/Inputs/In/nComState <-> WcState/WcState
//     Enc/Inputs/In/nDataIn1 <-> FB Inputs Channel 2/Position
//     Enc/Inputs/In/nDataIn1 <-> FB Inputs Channel 1/Position
//     Enc/Inputs/In/nState1 @bit 12 <-> FB Inputs Channel 2/Status/Diag
//     Enc/Inputs/In/nState1 @bit 12 <-> FB Inputs Channel 1/Status/Diag
//     Enc/Inputs/In/nState1 @bit 1 <-> FB Inputs Channel 2/Status/Error
//     Enc/Inputs/In/nState1 @bit 1 <-> FB Inputs Channel 1/Status/Error
//     Enc/Inputs/In/nState1 @bit 14 <-> FB Inputs Channel 2/Status/Input cycle counter
//     Enc/Inputs/In/nState1 @bit 14 <-> FB Inputs Channel 1/Status/Input cycle counter
//     Enc/Inputs/In/nState1 @bit 2 <-> FB Inputs Channel 2/Status/Ready
//     Enc/Inputs/In/nState1 @bit 2 <-> FB Inputs Channel 1/Status/Ready
//     Enc/Inputs/In/nState1 @bit 13 <-> FB Inputs Channel 2/Status/TxPDO State
//     Enc/Inputs/In/nState1 @bit 13 <-> FB Inputs Channel 1/Status/TxPDO State
//     Enc/Inputs/In/nState1 <-> FB Inputs Channel 2/Status/Warning
//     Enc/Inputs/In/nState1 <-> FB Inputs Channel 1/Status/Warning
//   (this object) <-> PLC Rail (EtherCAT)/Power (EK1200)/Fiber Coupler (EK1521-0010)/Term 123 (EK1100)/Term 131 (EK1122)/PF1K2-WFS (EK1100)/PF1K2-EL7041-E1
//     Drive/Inputs/In/nState1 @bit 3 <-> STM Status/Status/Error
//     Drive/Inputs/In/nState1 @bit 5 <-> STM Status/Status/Moving negative
//     Drive/Inputs/In/nState1 @bit 4 <-> STM Status/Status/Moving positive
//     Drive/Inputs/In/nState1 @bit 1 <-> STM Status/Status/Ready
//     Drive/Inputs/In/nState1 <-> STM Status/Status/Ready to enable
//     Drive/Inputs/In/nState1 @bit 6 <-> STM Status/Status/Torque reduced
//     Drive/Inputs/In/nState1 @bit 2 <-> STM Status/Status/Warning
//     Drive/Inputs/In/nState2 @bit 3 <-> STM Status/Status/Digital input 1
//     Drive/Inputs/In/nState2 @bit 4 <-> STM Status/Status/Digital input 2
//     Drive/Inputs/In/nState2 @bit 5 <-> STM Status/Status/Sync error
//     Drive/Inputs/In/nState2 @bit 7 <-> STM Status/Status/TxPDO Toggle
//     Drive/Inputs/In/nState4 @bit 1 <-> WcState/InputToggle
//     Drive/Inputs/In/nState4 <-> WcState/WcState
//     Drive/Outputs/Out/nCtrl1 <-> STM Control/Control/Enable
//     Drive/Outputs/Out/nCtrl1 @bit 2 <-> STM Control/Control/Reduce torque
//     Drive/Outputs/Out/nCtrl1 @bit 1 <-> STM Control/Control/Reset
//     Drive/Outputs/Out/nDataOut2[0] <-> STM Velocity/Velocity
//   (this object) <-> PLC Rail (EtherCAT)/Power (EK1200)/Fiber Coupler (EK1521-0010)/Term 123 (EK1100)/Term 131 (EK1122)/PF1K2-WFS (EK1100)/PF1K2-EL7041-E2
//     Drive/Inputs/In/nState1 @bit 3 <-> STM Status/Status/Error
//     Drive/Inputs/In/nState1 @bit 5 <-> STM Status/Status/Moving negative
//     Drive/Inputs/In/nState1 @bit 4 <-> STM Status/Status/Moving positive
//     Drive/Inputs/In/nState1 @bit 1 <-> STM Status/Status/Ready
//     Drive/Inputs/In/nState1 <-> STM Status/Status/Ready to enable
//     Drive/Inputs/In/nState1 @bit 6 <-> STM Status/Status/Torque reduced
//     Drive/Inputs/In/nState1 @bit 2 <-> STM Status/Status/Warning
//     Drive/Inputs/In/nState2 @bit 3 <-> STM Status/Status/Digital input 1
//     Drive/Inputs/In/nState2 @bit 4 <-> STM Status/Status/Digital input 2
//     Drive/Inputs/In/nState2 @bit 5 <-> STM Status/Status/Sync error
//     Drive/Inputs/In/nState2 @bit 7 <-> STM Status/Status/TxPDO Toggle
//     Drive/Inputs/In/nState4 @bit 1 <-> WcState/InputToggle
//     Drive/Inputs/In/nState4 <-> WcState/WcState
//     Drive/Outputs/Out/nCtrl1 <-> STM Control/Control/Enable
//     Drive/Outputs/Out/nCtrl1 @bit 2 <-> STM Control/Control/Reduce torque
//     Drive/Outputs/Out/nCtrl1 @bit 1 <-> STM Control/Control/Reset
//     Drive/Outputs/Out/nDataOut2[0] <-> STM Velocity/Velocity
//   (this object) <-> PLC Rail (EtherCAT)/Power (EK1200)/Fiber Coupler (EK1521-0010)/Term 123 (EK1100)/Term 140 (EK1122)/TM2K2-K2B (EK1100)/TM2K2-EL5042-E3
//     Enc/Inputs/In/nComState @bit 1 <-> WcState/InputToggle
//     Enc/Inputs/In/nComState <-> WcState/WcState
//     Enc/Inputs/In/nDataIn1 <-> FB Inputs Channel 1/Position
//     Enc/Inputs/In/nDataIn1 <-> FB Inputs Channel 2/Position
//     Enc/Inputs/In/nState1 @bit 12 <-> FB Inputs Channel 1/Status/Diag
//     Enc/Inputs/In/nState1 @bit 12 <-> FB Inputs Channel 2/Status/Diag
//     Enc/Inputs/In/nState1 @bit 1 <-> FB Inputs Channel 1/Status/Error
//     Enc/Inputs/In/nState1 @bit 1 <-> FB Inputs Channel 2/Status/Error
//     Enc/Inputs/In/nState1 @bit 14 <-> FB Inputs Channel 1/Status/Input cycle counter
//     Enc/Inputs/In/nState1 @bit 14 <-> FB Inputs Channel 2/Status/Input cycle counter
//     Enc/Inputs/In/nState1 @bit 2 <-> FB Inputs Channel 1/Status/Ready
//     Enc/Inputs/In/nState1 @bit 2 <-> FB Inputs Channel 2/Status/Ready
//     Enc/Inputs/In/nState1 @bit 13 <-> FB Inputs Channel 1/Status/TxPDO State
//     Enc/Inputs/In/nState1 @bit 13 <-> FB Inputs Channel 2/Status/TxPDO State
//     Enc/Inputs/In/nState1 <-> FB Inputs Channel 1/Status/Warning
//     Enc/Inputs/In/nState1 <-> FB Inputs Channel 2/Status/Warning
//   (this object) <-> PLC Rail (EtherCAT)/Power (EK1200)/Fiber Coupler (EK1521-0010)/Term 123 (EK1100)/Term 140 (EK1122)/TM2K2-K2B (EK1100)/TM2K2-EL7041-E1
//     Drive/Inputs/In/nState1 @bit 3 <-> STM Status/Status/Error
//     Drive/Inputs/In/nState1 @bit 5 <-> STM Status/Status/Moving negative
//     Drive/Inputs/In/nState1 @bit 4 <-> STM Status/Status/Moving positive
//     Drive/Inputs/In/nState1 @bit 1 <-> STM Status/Status/Ready
//     Drive/Inputs/In/nState1 <-> STM Status/Status/Ready to enable
//     Drive/Inputs/In/nState1 @bit 6 <-> STM Status/Status/Torque reduced
//     Drive/Inputs/In/nState1 @bit 2 <-> STM Status/Status/Warning
//     Drive/Inputs/In/nState2 @bit 3 <-> STM Status/Status/Digital input 1
//     Drive/Inputs/In/nState2 @bit 4 <-> STM Status/Status/Digital input 2
//     Drive/Inputs/In/nState2 @bit 5 <-> STM Status/Status/Sync error
//     Drive/Inputs/In/nState2 @bit 7 <-> STM Status/Status/TxPDO Toggle
//     Drive/Inputs/In/nState4 @bit 1 <-> WcState/InputToggle
//     Drive/Inputs/In/nState4 <-> WcState/WcState
//     Drive/Outputs/Out/nCtrl1 <-> STM Control/Control/Enable
//     Drive/Outputs/Out/nCtrl1 @bit 2 <-> STM Control/Control/Reduce torque
//     Drive/Outputs/Out/nCtrl1 @bit 1 <-> STM Control/Control/Reset
//     Drive/Outputs/Out/nDataOut2[0] <-> STM Velocity/Velocity
//   (this object) <-> PLC Rail (EtherCAT)/Power (EK1200)/Fiber Coupler (EK1521-0010)/Term 123 (EK1100)/Term 140 (EK1122)/TM2K2-K2B (EK1100)/TM2K2-EL7041-E2
//     Drive/Inputs/In/nState1 @bit 3 <-> STM Status/Status/Error
//     Drive/Inputs/In/nState1 @bit 5 <-> STM Status/Status/Moving negative
//     Drive/Inputs/In/nState1 @bit 4 <-> STM Status/Status/Moving positive
//     Drive/Inputs/In/nState1 @bit 1 <-> STM Status/Status/Ready
//     Drive/Inputs/In/nState1 <-> STM Status/Status/Ready to enable
//     Drive/Inputs/In/nState1 @bit 6 <-> STM Status/Status/Torque reduced
//     Drive/Inputs/In/nState1 @bit 2 <-> STM Status/Status/Warning
//     Drive/Inputs/In/nState2 @bit 3 <-> STM Status/Status/Digital input 1
//     Drive/Inputs/In/nState2 @bit 4 <-> STM Status/Status/Digital input 2
//     Drive/Inputs/In/nState2 @bit 5 <-> STM Status/Status/Sync error
//     Drive/Inputs/In/nState2 @bit 7 <-> STM Status/Status/TxPDO Toggle
//     Drive/Inputs/In/nState4 @bit 1 <-> WcState/InputToggle
//     Drive/Inputs/In/nState4 <-> WcState/WcState
//     Drive/Outputs/Out/nCtrl1 <-> STM Control/Control/Enable
//     Drive/Outputs/Out/nCtrl1 @bit 2 <-> STM Control/Control/Reduce torque
//     Drive/Outputs/Out/nCtrl1 @bit 1 <-> STM Control/Control/Reset
//     Drive/Outputs/Out/nDataOut2[0] <-> STM Velocity/Velocity
//   (this object) <-> PLC Rail (EtherCAT)/Power (EK1200)/Fiber Coupler (EK1521-0010)/Term 123 (EK1100)/Term 155 (EK1122)/AT2K2-SOLID (EK1100)/AT2K2-EL5042-01
//     Enc/Inputs/In/nComState @bit 1 <-> WcState/InputToggle
//     Enc/Inputs/In/nComState <-> WcState/WcState
//     Enc/Inputs/In/nDataIn1 <-> FB Inputs Channel 1/Position
//     Enc/Inputs/In/nDataIn1 <-> FB Inputs Channel 2/Position
//     Enc/Inputs/In/nState1 @bit 12 <-> FB Inputs Channel 1/Status/Diag
//     Enc/Inputs/In/nState1 @bit 12 <-> FB Inputs Channel 2/Status/Diag
//     Enc/Inputs/In/nState1 @bit 1 <-> FB Inputs Channel 1/Status/Error
//     Enc/Inputs/In/nState1 @bit 1 <-> FB Inputs Channel 2/Status/Error
//     Enc/Inputs/In/nState1 @bit 14 <-> FB Inputs Channel 1/Status/Input cycle counter
//     Enc/Inputs/In/nState1 @bit 14 <-> FB Inputs Channel 2/Status/Input cycle counter
//     Enc/Inputs/In/nState1 @bit 2 <-> FB Inputs Channel 1/Status/Ready
//     Enc/Inputs/In/nState1 @bit 2 <-> FB Inputs Channel 2/Status/Ready
//     Enc/Inputs/In/nState1 @bit 13 <-> FB Inputs Channel 1/Status/TxPDO State
//     Enc/Inputs/In/nState1 @bit 13 <-> FB Inputs Channel 2/Status/TxPDO State
//     Enc/Inputs/In/nState1 <-> FB Inputs Channel 1/Status/Warning
//     Enc/Inputs/In/nState1 <-> FB Inputs Channel 2/Status/Warning
//   (this object) <-> PLC Rail (EtherCAT)/Power (EK1200)/Fiber Coupler (EK1521-0010)/Term 123 (EK1100)/Term 155 (EK1122)/AT2K2-SOLID (EK1100)/AT2K2-EL7047-01
//     Drive/Inputs/In/nState1 @bit 3 <-> STM Status/Status/Error
//     Drive/Inputs/In/nState1 @bit 7 <-> STM Status/Status/Motor stall
//     Drive/Inputs/In/nState1 @bit 5 <-> STM Status/Status/Moving negative
//     Drive/Inputs/In/nState1 @bit 4 <-> STM Status/Status/Moving positive
//     Drive/Inputs/In/nState1 @bit 1 <-> STM Status/Status/Ready
//     Drive/Inputs/In/nState1 <-> STM Status/Status/Ready to enable
//     Drive/Inputs/In/nState1 @bit 6 <-> STM Status/Status/Torque reduced
//     Drive/Inputs/In/nState1 @bit 2 <-> STM Status/Status/Warning
//     Drive/Inputs/In/nState2 @bit 3 <-> STM Status/Status/Digital input 1
//     Drive/Inputs/In/nState2 @bit 4 <-> STM Status/Status/Digital input 2
//     Drive/Inputs/In/nState2 @bit 5 <-> STM Status/Status/Sync error
//     Drive/Inputs/In/nState2 @bit 7 <-> STM Status/Status/TxPDO Toggle
//     Drive/Inputs/In/nState4 @bit 1 <-> WcState/InputToggle
//     Drive/Inputs/In/nState4 <-> WcState/WcState
//     Drive/Outputs/Out/nCtrl1 <-> STM Control/Control/Enable
//     Drive/Outputs/Out/nCtrl1 @bit 2 <-> STM Control/Control/Reduce torque
//     Drive/Outputs/Out/nCtrl1 @bit 1 <-> STM Control/Control/Reset
//     Drive/Outputs/Out/nCtrl2 @bit 3 <-> STM Control/Control/Digital output 1
//     Drive/Outputs/Out/nDataOut2[0] <-> STM Velocity/Velocity
//   (this object) <-> PLC Rail (EtherCAT)/Power (EK1200)/Fiber Coupler (EK1521-0010)/Term 123 (EK1100)/Term 155 (EK1122)/AT2K2-SOLID (EK1100)/AT2K2-EL7047-02
//     Drive/Inputs/In/nState1 @bit 3 <-> STM Status/Status/Error
//     Drive/Inputs/In/nState1 @bit 7 <-> STM Status/Status/Motor stall
//     Drive/Inputs/In/nState1 @bit 5 <-> STM Status/Status/Moving negative
//     Drive/Inputs/In/nState1 @bit 4 <-> STM Status/Status/Moving positive
//     Drive/Inputs/In/nState1 @bit 1 <-> STM Status/Status/Ready
//     Drive/Inputs/In/nState1 <-> STM Status/Status/Ready to enable
//     Drive/Inputs/In/nState1 @bit 6 <-> STM Status/Status/Torque reduced
//     Drive/Inputs/In/nState1 @bit 2 <-> STM Status/Status/Warning
//     Drive/Inputs/In/nState2 @bit 3 <-> STM Status/Status/Digital input 1
//     Drive/Inputs/In/nState2 @bit 4 <-> STM Status/Status/Digital input 2
//     Drive/Inputs/In/nState2 @bit 5 <-> STM Status/Status/Sync error
//     Drive/Inputs/In/nState2 @bit 7 <-> STM Status/Status/TxPDO Toggle
//     Drive/Inputs/In/nState4 @bit 1 <-> WcState/InputToggle
//     Drive/Inputs/In/nState4 <-> WcState/WcState
//     Drive/Outputs/Out/nCtrl1 <-> STM Control/Control/Enable
//     Drive/Outputs/Out/nCtrl1 @bit 2 <-> STM Control/Control/Reduce torque
//     Drive/Outputs/Out/nCtrl1 @bit 1 <-> STM Control/Control/Reset
//     Drive/Outputs/Out/nCtrl2 @bit 3 <-> STM Control/Control/Digital output 1
//     Drive/Outputs/Out/nDataOut2[0] <-> STM Velocity/Velocity
//   (this object) <-> PLC Rail (EtherCAT)/Power (EK1200)/Fiber Coupler (EK1521-0010)/Term 123 (EK1100)/Term 155 (EK1122)/AT2K2-SOLID (EK1100)/AT2K2-EL5042-02
//     Enc/Inputs/In/nComState @bit 1 <-> WcState/InputToggle
//     Enc/Inputs/In/nComState <-> WcState/WcState
//     Enc/Inputs/In/nDataIn1 <-> FB Inputs Channel 1/Position
//     Enc/Inputs/In/nDataIn1 <-> FB Inputs Channel 2/Position
//     Enc/Inputs/In/nState1 @bit 12 <-> FB Inputs Channel 1/Status/Diag
//     Enc/Inputs/In/nState1 @bit 12 <-> FB Inputs Channel 2/Status/Diag
//     Enc/Inputs/In/nState1 @bit 1 <-> FB Inputs Channel 1/Status/Error
//     Enc/Inputs/In/nState1 @bit 1 <-> FB Inputs Channel 2/Status/Error
//     Enc/Inputs/In/nState1 @bit 14 <-> FB Inputs Channel 1/Status/Input cycle counter
//     Enc/Inputs/In/nState1 @bit 14 <-> FB Inputs Channel 2/Status/Input cycle counter
//     Enc/Inputs/In/nState1 @bit 2 <-> FB Inputs Channel 1/Status/Ready
//     Enc/Inputs/In/nState1 @bit 2 <-> FB Inputs Channel 2/Status/Ready
//     Enc/Inputs/In/nState1 @bit 13 <-> FB Inputs Channel 1/Status/TxPDO State
//     Enc/Inputs/In/nState1 @bit 13 <-> FB Inputs Channel 2/Status/TxPDO State
//     Enc/Inputs/In/nState1 <-> FB Inputs Channel 1/Status/Warning
//     Enc/Inputs/In/nState1 <-> FB Inputs Channel 2/Status/Warning
//   (this object) <-> PLC Rail (EtherCAT)/Power (EK1200)/Fiber Coupler (EK1521-0010)/Term 123 (EK1100)/Term 155 (EK1122)/AT2K2-SOLID (EK1100)/AT2K2-EL7047-03
//     Drive/Inputs/In/nState1 @bit 3 <-> STM Status/Status/Error
//     Drive/Inputs/In/nState1 @bit 7 <-> STM Status/Status/Motor stall
//     Drive/Inputs/In/nState1 @bit 5 <-> STM Status/Status/Moving negative
//     Drive/Inputs/In/nState1 @bit 4 <-> STM Status/Status/Moving positive
//     Drive/Inputs/In/nState1 @bit 1 <-> STM Status/Status/Ready
//     Drive/Inputs/In/nState1 <-> STM Status/Status/Ready to enable
//     Drive/Inputs/In/nState1 @bit 6 <-> STM Status/Status/Torque reduced
//     Drive/Inputs/In/nState1 @bit 2 <-> STM Status/Status/Warning
//     Drive/Inputs/In/nState2 @bit 3 <-> STM Status/Status/Digital input 1
//     Drive/Inputs/In/nState2 @bit 4 <-> STM Status/Status/Digital input 2
//     Drive/Inputs/In/nState2 @bit 5 <-> STM Status/Status/Sync error
//     Drive/Inputs/In/nState2 @bit 7 <-> STM Status/Status/TxPDO Toggle
//     Drive/Inputs/In/nState4 @bit 1 <-> WcState/InputToggle
//     Drive/Inputs/In/nState4 <-> WcState/WcState
//     Drive/Outputs/Out/nCtrl1 <-> STM Control/Control/Enable
//     Drive/Outputs/Out/nCtrl1 @bit 2 <-> STM Control/Control/Reduce torque
//     Drive/Outputs/Out/nCtrl1 @bit 1 <-> STM Control/Control/Reset
//     Drive/Outputs/Out/nCtrl2 @bit 3 <-> STM Control/Control/Digital output 1
//     Drive/Outputs/Out/nDataOut2[0] <-> STM Velocity/Velocity
//   (this object) <-> PLC Rail (EtherCAT)/Power (EK1200)/Fiber Coupler (EK1521-0010)/Term 123 (EK1100)/Term 155 (EK1122)/AT2K2-SOLID (EK1100)/AT2K2-EL7047-04
//     Drive/Inputs/In/nState1 @bit 3 <-> STM Status/Status/Error
//     Drive/Inputs/In/nState1 @bit 7 <-> STM Status/Status/Motor stall
//     Drive/Inputs/In/nState1 @bit 5 <-> STM Status/Status/Moving negative
//     Drive/Inputs/In/nState1 @bit 4 <-> STM Status/Status/Moving positive
//     Drive/Inputs/In/nState1 @bit 1 <-> STM Status/Status/Ready
//     Drive/Inputs/In/nState1 <-> STM Status/Status/Ready to enable
//     Drive/Inputs/In/nState1 @bit 6 <-> STM Status/Status/Torque reduced
//     Drive/Inputs/In/nState1 @bit 2 <-> STM Status/Status/Warning
//     Drive/Inputs/In/nState2 @bit 3 <-> STM Status/Status/Digital input 1
//     Drive/Inputs/In/nState2 @bit 4 <-> STM Status/Status/Digital input 2
//     Drive/Inputs/In/nState2 @bit 5 <-> STM Status/Status/Sync error
//     Drive/Inputs/In/nState2 @bit 7 <-> STM Status/Status/TxPDO Toggle
//     Drive/Inputs/In/nState4 @bit 1 <-> WcState/InputToggle
//     Drive/Inputs/In/nState4 <-> WcState/WcState
//     Drive/Outputs/Out/nCtrl1 <-> STM Control/Control/Enable
//     Drive/Outputs/Out/nCtrl1 @bit 2 <-> STM Control/Control/Reduce torque
//     Drive/Outputs/Out/nCtrl1 @bit 1 <-> STM Control/Control/Reset
//     Drive/Outputs/Out/nCtrl2 @bit 3 <-> STM Control/Control/Digital output 1
//     Drive/Outputs/Out/nDataOut2[0] <-> STM Velocity/Velocity
//   (this object) <-> PLC Rail (EtherCAT)/Power (EK1200)/Fiber Coupler (EK1521-0010)/Term 123 (EK1100)/Term 155 (EK1122)/LI3K2-K2B (EK1100)/LI3K2-EL5042-E2
//     Enc/Inputs/In/nComState @bit 1 <-> WcState/InputToggle
//     Enc/Inputs/In/nComState <-> WcState/WcState
//     Enc/Inputs/In/nDataIn1 <-> FB Inputs Channel 1/Position
//     Enc/Inputs/In/nState1 @bit 12 <-> FB Inputs Channel 1/Status/Diag
//     Enc/Inputs/In/nState1 @bit 1 <-> FB Inputs Channel 1/Status/Error
//     Enc/Inputs/In/nState1 @bit 14 <-> FB Inputs Channel 1/Status/Input cycle counter
//     Enc/Inputs/In/nState1 @bit 2 <-> FB Inputs Channel 1/Status/Ready
//     Enc/Inputs/In/nState1 @bit 13 <-> FB Inputs Channel 1/Status/TxPDO State
//     Enc/Inputs/In/nState1 <-> FB Inputs Channel 1/Status/Warning
//   (this object) <-> PLC Rail (EtherCAT)/Power (EK1200)/Fiber Coupler (EK1521-0010)/Term 123 (EK1100)/Term 155 (EK1122)/LI3K2-K2B (EK1100)/LI3K2-EL7041-E1
//     Drive/Inputs/In/nState1 @bit 3 <-> STM Status/Status/Error
//     Drive/Inputs/In/nState1 @bit 5 <-> STM Status/Status/Moving negative
//     Drive/Inputs/In/nState1 @bit 4 <-> STM Status/Status/Moving positive
//     Drive/Inputs/In/nState1 @bit 1 <-> STM Status/Status/Ready
//     Drive/Inputs/In/nState1 <-> STM Status/Status/Ready to enable
//     Drive/Inputs/In/nState1 @bit 6 <-> STM Status/Status/Torque reduced
//     Drive/Inputs/In/nState1 @bit 2 <-> STM Status/Status/Warning
//     Drive/Inputs/In/nState2 @bit 3 <-> STM Status/Status/Digital input 1
//     Drive/Inputs/In/nState2 @bit 4 <-> STM Status/Status/Digital input 2
//     Drive/Inputs/In/nState2 @bit 5 <-> STM Status/Status/Sync error
//     Drive/Inputs/In/nState2 @bit 7 <-> STM Status/Status/TxPDO Toggle
//     Drive/Inputs/In/nState4 @bit 1 <-> WcState/InputToggle
//     Drive/Inputs/In/nState4 <-> WcState/WcState
//     Drive/Outputs/Out/nCtrl1 <-> STM Control/Control/Enable
//     Drive/Outputs/Out/nCtrl1 @bit 2 <-> STM Control/Control/Reduce torque
//     Drive/Outputs/Out/nCtrl1 @bit 1 <-> STM Control/Control/Reset
//     Drive/Outputs/Out/nDataOut2[0] <-> STM Velocity/Velocity
//   (this object) <-> PLC Rail (EtherCAT)/Power (EK1200)/Fiber Coupler (EK1521-0010)/Term 123 (EK1100)/Term 156 (EK1122)/PF2K2-WFS (EK1100)/PF2K2-EL5042-E3
//     Enc/Inputs/In/nComState @bit 1 <-> WcState/InputToggle
//     Enc/Inputs/In/nComState <-> WcState/WcState
//     Enc/Inputs/In/nDataIn1 <-> FB Inputs Channel 2/Position
//     Enc/Inputs/In/nDataIn1 <-> FB Inputs Channel 1/Position
//     Enc/Inputs/In/nState1 @bit 12 <-> FB Inputs Channel 2/Status/Diag
//     Enc/Inputs/In/nState1 @bit 12 <-> FB Inputs Channel 1/Status/Diag
//     Enc/Inputs/In/nState1 @bit 1 <-> FB Inputs Channel 2/Status/Error
//     Enc/Inputs/In/nState1 @bit 1 <-> FB Inputs Channel 1/Status/Error
//     Enc/Inputs/In/nState1 @bit 14 <-> FB Inputs Channel 2/Status/Input cycle counter
//     Enc/Inputs/In/nState1 @bit 14 <-> FB Inputs Channel 1/Status/Input cycle counter
//     Enc/Inputs/In/nState1 @bit 2 <-> FB Inputs Channel 2/Status/Ready
//     Enc/Inputs/In/nState1 @bit 2 <-> FB Inputs Channel 1/Status/Ready
//     Enc/Inputs/In/nState1 @bit 13 <-> FB Inputs Channel 2/Status/TxPDO State
//     Enc/Inputs/In/nState1 @bit 13 <-> FB Inputs Channel 1/Status/TxPDO State
//     Enc/Inputs/In/nState1 <-> FB Inputs Channel 2/Status/Warning
//     Enc/Inputs/In/nState1 <-> FB Inputs Channel 1/Status/Warning
//   (this object) <-> PLC Rail (EtherCAT)/Power (EK1200)/Fiber Coupler (EK1521-0010)/Term 123 (EK1100)/Term 156 (EK1122)/PF2K2-WFS (EK1100)/PF2K2-EL7041-E1
//     Drive/Inputs/In/nState1 @bit 3 <-> STM Status/Status/Error
//     Drive/Inputs/In/nState1 @bit 5 <-> STM Status/Status/Moving negative
//     Drive/Inputs/In/nState1 @bit 4 <-> STM Status/Status/Moving positive
//     Drive/Inputs/In/nState1 @bit 1 <-> STM Status/Status/Ready
//     Drive/Inputs/In/nState1 <-> STM Status/Status/Ready to enable
//     Drive/Inputs/In/nState1 @bit 6 <-> STM Status/Status/Torque reduced
//     Drive/Inputs/In/nState1 @bit 2 <-> STM Status/Status/Warning
//     Drive/Inputs/In/nState2 @bit 3 <-> STM Status/Status/Digital input 1
//     Drive/Inputs/In/nState2 @bit 4 <-> STM Status/Status/Digital input 2
//     Drive/Inputs/In/nState2 @bit 5 <-> STM Status/Status/Sync error
//     Drive/Inputs/In/nState2 @bit 7 <-> STM Status/Status/TxPDO Toggle
//     Drive/Inputs/In/nState4 @bit 1 <-> WcState/InputToggle
//     Drive/Inputs/In/nState4 <-> WcState/WcState
//     Drive/Outputs/Out/nCtrl1 <-> STM Control/Control/Enable
//     Drive/Outputs/Out/nCtrl1 @bit 2 <-> STM Control/Control/Reduce torque
//     Drive/Outputs/Out/nCtrl1 @bit 1 <-> STM Control/Control/Reset
//     Drive/Outputs/Out/nDataOut2[0] <-> STM Velocity/Velocity
//   (this object) <-> PLC Rail (EtherCAT)/Power (EK1200)/Fiber Coupler (EK1521-0010)/Term 123 (EK1100)/Term 156 (EK1122)/PF2K2-WFS (EK1100)/PF2K2-EL7041-E2
//     Drive/Inputs/In/nState1 @bit 3 <-> STM Status/Status/Error
//     Drive/Inputs/In/nState1 @bit 5 <-> STM Status/Status/Moving negative
//     Drive/Inputs/In/nState1 @bit 4 <-> STM Status/Status/Moving positive
//     Drive/Inputs/In/nState1 @bit 1 <-> STM Status/Status/Ready
//     Drive/Inputs/In/nState1 <-> STM Status/Status/Ready to enable
//     Drive/Inputs/In/nState1 @bit 6 <-> STM Status/Status/Torque reduced
//     Drive/Inputs/In/nState1 @bit 2 <-> STM Status/Status/Warning
//     Drive/Inputs/In/nState2 @bit 3 <-> STM Status/Status/Digital input 1
//     Drive/Inputs/In/nState2 @bit 4 <-> STM Status/Status/Digital input 2
//     Drive/Inputs/In/nState2 @bit 5 <-> STM Status/Status/Sync error
//     Drive/Inputs/In/nState2 @bit 7 <-> STM Status/Status/TxPDO Toggle
//     Drive/Inputs/In/nState4 @bit 1 <-> WcState/InputToggle
//     Drive/Inputs/In/nState4 <-> WcState/WcState
//     Drive/Outputs/Out/nCtrl1 <-> STM Control/Control/Enable
//     Drive/Outputs/Out/nCtrl1 @bit 2 <-> STM Control/Control/Reduce torque
//     Drive/Outputs/Out/nCtrl1 @bit 1 <-> STM Control/Control/Reset
//     Drive/Outputs/Out/nDataOut2[0] <-> STM Velocity/Velocity
//   (this object) <-> PLC Rail (EtherCAT)/Power (EK1200)/Fiber Coupler (EK1521-0010)/Term 123 (EK1100)/Term 156 (EK1122)/IM6K2-PPM (EK1100)/IM6K2-EL5042-E2
//     Enc/Inputs/In/nComState @bit 1 <-> WcState/InputToggle
//     Enc/Inputs/In/nComState <-> WcState/WcState
//     Enc/Inputs/In/nDataIn1 <-> FB Inputs Channel 1/Position
//     Enc/Inputs/In/nState1 @bit 12 <-> FB Inputs Channel 1/Status/Diag
//     Enc/Inputs/In/nState1 @bit 1 <-> FB Inputs Channel 1/Status/Error
//     Enc/Inputs/In/nState1 @bit 14 <-> FB Inputs Channel 1/Status/Input cycle counter
//     Enc/Inputs/In/nState1 @bit 2 <-> FB Inputs Channel 1/Status/Ready
//     Enc/Inputs/In/nState1 @bit 13 <-> FB Inputs Channel 1/Status/TxPDO State
//     Enc/Inputs/In/nState1 <-> FB Inputs Channel 1/Status/Warning
//   (this object) <-> PLC Rail (EtherCAT)/Power (EK1200)/Fiber Coupler (EK1521-0010)/Term 123 (EK1100)/Term 156 (EK1122)/IM6K2-PPM (EK1100)/IM6K2-EL7041-E1
//     Drive/Inputs/In/nState1 @bit 3 <-> STM Status/Status/Error
//     Drive/Inputs/In/nState1 @bit 5 <-> STM Status/Status/Moving negative
//     Drive/Inputs/In/nState1 @bit 4 <-> STM Status/Status/Moving positive
//     Drive/Inputs/In/nState1 @bit 1 <-> STM Status/Status/Ready
//     Drive/Inputs/In/nState1 <-> STM Status/Status/Ready to enable
//     Drive/Inputs/In/nState1 @bit 6 <-> STM Status/Status/Torque reduced
//     Drive/Inputs/In/nState1 @bit 2 <-> STM Status/Status/Warning
//     Drive/Inputs/In/nState2 @bit 3 <-> STM Status/Status/Digital input 1
//     Drive/Inputs/In/nState2 @bit 4 <-> STM Status/Status/Digital input 2
//     Drive/Inputs/In/nState2 @bit 5 <-> STM Status/Status/Sync error
//     Drive/Inputs/In/nState2 @bit 7 <-> STM Status/Status/TxPDO Toggle
//     Drive/Inputs/In/nState4 @bit 1 <-> WcState/InputToggle
//     Drive/Inputs/In/nState4 <-> WcState/WcState
//     Drive/Outputs/Out/nCtrl1 <-> STM Control/Control/Enable
//     Drive/Outputs/Out/nCtrl1 @bit 2 <-> STM Control/Control/Reduce torque
//     Drive/Outputs/Out/nCtrl1 @bit 1 <-> STM Control/Control/Reset
//     Drive/Outputs/Out/nDataOut2[0] <-> STM Velocity/Velocity
//   (this object) <-> PLC Rail (EtherCAT)/Power (EK1200)/Fiber Coupler (EK1521-0010)/Term 123 (EK1100)/Term 73 (EK1122)/PAX-DRL-02 (EK1100)/PAX-EL5042-E16
//     Enc/Inputs/In/nComState @bit 1 <-> WcState/InputToggle
//     Enc/Inputs/In/nComState <-> WcState/WcState
//     Enc/Inputs/In/nDataIn1 <-> FB Inputs Channel 2/Position
//     Enc/Inputs/In/nDataIn1 <-> FB Inputs Channel 1/Position
//     Enc/Inputs/In/nState1 @bit 12 <-> FB Inputs Channel 2/Status/Diag
//     Enc/Inputs/In/nState1 @bit 12 <-> FB Inputs Channel 1/Status/Diag
